# B&R Automation Studio project NAEUL004C00R13L518F00 (part 19)

#### Act_OptP0931MagConv2FB.st
```iecst
ACTION Act_OptP0931MagConv2FB:

	//Magazine Conveyor
	IF tyP0931MagConv2.tyFB.tyBtnStop.bRtCompl = TRUE THEN
		eMagConv2Clp2Act	:= MagConv2ClpActStop;

		IF p_eMagConv2Clp2Stat = MagConv2ClpActStop AND p_eMagConv2Clp2Status = Done THEN
			eMagConv2Clp2Act	:= MagConv2ClpActIdle;

			tyP0931MagConv2.tyFB.tyBtnEnt.bRtCompl	:= FALSE;
			tyP0931MagConv2.tyFB.tyBtnEnt.bValue	:= FALSE;
			tyP0931MagConv2.tyFB.tyBtnEnt.bRtLk		:= FALSE;

			tyP0931MagConv2.tyFB.tyBtnExit.bRtCompl	:= FALSE;
			tyP0931MagConv2.tyFB.tyBtnExit.bValue	:= FALSE;
			tyP0931MagConv2.tyFB.tyBtnExit.bRtLk	:= FALSE;

			tyP0931MagConv2.tyFB.tyBtnStop.bRtCompl	:= FALSE;
			tyP0931MagConv2.tyFB.tyBtnStop.bValue	:= TRUE;
			tyP0931MagConv2.tyFB.tyBtnStop.bRtLk	:= TRUE;
		END_IF

	ELSIF tyP0931MagConv2.tyFB.tyBtnEnt.bRtCompl = TRUE THEN
		tyP0931MagConv2.tyFB.tyBtnEnt.bValue	:= TRUE;
		tyP0931MagConv2.tyFB.tyBtnEnt.bRtLk		:= TRUE;

		tyP0931MagConv2.tyFB.tyBtnStop.bValue	:= FALSE;
		tyP0931MagConv2.tyFB.tyBtnStop.bRtLk	:= FALSE;

		eMagConv2Clp2Act	:= MagConv2ClpActEnt;

		IF p_eMagConv2Clp2Stat = MagConv2ClpActEnt AND p_eMagConv2Clp2Status = Done THEN
			eMagConv2Clp2Act	:= MagConv2ClpActIdle;

			tyP0931MagConv2.tyFB.tyBtnEnt.bRtCompl	:= FALSE;

			tyP0931MagConv2.tyFB.tyBtnEnt.bValue	:= FALSE;
			tyP0931MagConv2.tyFB.tyBtnEnt.bRtLk		:= FALSE;

			tyP0931MagConv2.tyFB.tyBtnStop.bValue	:= TRUE;
			tyP0931MagConv2.tyFB.tyBtnStop.bRtLk	:= TRUE;
		END_IF

	ELSIF (p_eMagConv2Clp2Stat = MagConv2ClpActPreExit AND p_eMagConv2Clp2Status = Done) THEN
		eMagConv2Clp2Act	:= MagConv2ClpActIdle;

		tyP0931MagConv2.tyFB.tyBtnExit.bRtCompl	:= FALSE;

		tyP0931MagConv2.tyFB.tyBtnExit.bValue	:= FALSE;
		tyP0931MagConv2.tyFB.tyBtnExit.bRtLk	:= FALSE;

		tyP0931MagConv2.tyFB.tyBtnStop.bValue	:= TRUE;
		tyP0931MagConv2.tyFB.tyBtnStop.bRtLk	:= TRUE;

	ELSIF (p_eMagConv2Clp2Stat = MagConv2ClpActExit AND p_eMagConv2Clp2Status = Done) THEN
		eMagConv2Clp2Act	:= MagConv2ClpActIdle;

		tyP0931MagConv2.tyFB.tyBtnExit.bRtCompl	:= FALSE;

		tyP0931MagConv2.tyFB.tyBtnExit.bValue	:= FALSE;
		tyP0931MagConv2.tyFB.tyBtnExit.bRtLk	:= FALSE;

		tyP0931MagConv2.tyFB.tyBtnStop.bValue	:= TRUE;
		tyP0931MagConv2.tyFB.tyBtnStop.bRtLk	:= TRUE;

	ELSIF tyP0931MagConv2.tyFB.tyBtnExit.bRtCompl = TRUE THEN
		tyP0931MagConv2.tyFB.tyBtnExit.bRtCompl	:= FALSE;
		tyP0931MagConv2.tyFB.tyBtnExit.bValue	:= TRUE;
		tyP0931MagConv2.tyFB.tyBtnExit.bRtLk	:= TRUE;

		tyP0931MagConv2.tyFB.tyBtnStop.bValue	:= FALSE;
		tyP0931MagConv2.tyFB.tyBtnStop.bRtLk	:= FALSE;

		IF p_tyDI.bMagConvEntSen2  THEN
			eMagConv2Clp2Act	:= MagConv2ClpActExit;
		ELSE
			IF p_tyDI.bMagPresentSen2 THEN
				eMagConv2Clp2Act	:= MagConv2ClpActPreExit;
			ELSE
				eMagConv2Clp2Act	:= MagConv2ClpActExit;
			END_IF
		END_IF
	END_IF

	//Magazine Clamper
	IF tyP0931MagConv2.tyCom.tyBtnSwitch.bValue = FALSE THEN

		//Fixed
		IF tyP0931MagConv2.tyFB.tyBtnFixedUnclamp.bRtCompl = TRUE THEN
			tyP0931MagConv2.tyFB.tyBtnFixedUnclamp.bRtCompl	:= FALSE;

			tyP0931MagConv2.tyFB.tyBtnFixedUnclamp.bValue	:= TRUE;
			tyP0931MagConv2.tyFB.tyBtnFixedClamp.bValue		:= FALSE;

		ELSIF tyP0931MagConv2.tyFB.tyBtnFixedClamp.bRtCompl = TRUE THEN
			tyP0931MagConv2.tyFB.tyBtnFixedClamp.bRtCompl	:= FALSE;

			tyP0931MagConv2.tyFB.tyBtnFixedClamp.bValue		:= TRUE;
			tyP0931MagConv2.tyFB.tyBtnFixedUnclamp.bValue	:= FALSE;

		END_IF

		//Remote
		IF tyP0931MagConv2.tyFB.tyBtnRemoteUnclamp.bRtCompl = TRUE THEN
			tyP0931MagConv2.tyFB.tyBtnRemoteUnclamp.bRtCompl	:= FALSE;

			tyP0931MagConv2.tyFB.tyBtnRemoteUnclamp.bValue	:= TRUE;
			tyP0931MagConv2.tyFB.tyBtnRemoteClamp.bValue	:= FALSE;

		ELSIF tyP0931MagConv2.tyFB.tyBtnRemoteClamp.bRtCompl = TRUE THEN
			tyP0931MagConv2.tyFB.tyBtnRemoteClamp.bRtCompl	:= FALSE;

			tyP0931MagConv2.tyFB.tyBtnRemoteClamp.bValue	:= TRUE;
			tyP0931MagConv2.tyFB.tyBtnRemoteUnclamp.bValue	:= FALSE;

		END_IF

		//Selection
		IF tyP0931MagConv2.tyFB.tyBtnSelUnclamp.bRtCompl = TRUE THEN
			tyP0931MagConv2.tyFB.tyBtnSelUnclamp.bRtCompl	:= FALSE;

			tyP0931MagConv2.tyFB.tyBtnSelUnclamp.bValue	:= TRUE;
			tyP0931MagConv2.tyFB.tyBtnSelClamp.bValue	:= FALSE;

		ELSIF tyP0931MagConv2.tyFB.tyBtnSelClamp.bRtCompl = TRUE THEN
			tyP0931MagConv2.tyFB.tyBtnSelClamp.bRtCompl	:= FALSE;

			tyP0931MagConv2.tyFB.tyBtnSelClamp.bValue	:= TRUE;
			tyP0931MagConv2.tyFB.tyBtnSelUnclamp.bValue	:= FALSE;

		END_IF

		// Fixed Clamper
		IF tyP0931MagConv2.tyFB.tyBtnFixedUnclamp.bValue = TRUE THEN

			eMagConv2Clp2Act	:= MagConv2ClpActFixClprUnclamp;

			IF p_eMagConv2Clp2Stat = MagConv2ClpActFixClprUnclamp AND p_eMagConv2Clp2Status = Done THEN

				eMagConv2Clp2Act	:= MagConv2ClpActIdle;

				tyP0931MagConv2.tyFB.tyBtnFixedUnclamp.bValue	:= FALSE;

			ELSIF p_eMagConv2Clp2Status = Error THEN

				tyP0931MagConv2.tyFB.tyBtnFixedUnclamp.bValue	:= FALSE;

			END_IF

		ELSIF tyP0931MagConv2.tyFB.tyBtnFixedClamp.bValue = TRUE THEN
			eMagConv2Clp2Act	:= MagConv2ClpActFixClprClamp;

			IF p_eMagConv2Clp2Stat = MagConv2ClpActFixClprClamp AND p_eMagConv2Clp2Status = Done THEN

				eMagConv2Clp2Act	:= MagConv2ClpActIdle;

				tyP0931MagConv2.tyFB.tyBtnFixedClamp.bValue := FALSE;

			ELSIF p_eMagConv2Clp2Status = Error THEN
				tyP0931MagConv2.tyFB.tyBtnFixedClamp.bValue := FALSE;

			END_IF

		END_IF

		//Remote Clamper
		IF tyP0931MagConv2.tyFB.tyBtnRemoteUnclamp.bValue = TRUE THEN

			eMagConv2Clp2Act	:= MagConv2ClpActRmtClprUnclamp;

			IF p_eMagConv2Clp2Stat = MagConv2ClpActRmtClprUnclamp AND p_eMagConv2Clp2Status = Done THEN

				eMagConv2Clp2Act	:= MagConv2ClpActIdle;

				tyP0931MagConv2.tyFB.tyBtnRemoteUnclamp.bValue	:= FALSE;

			ELSIF p_eMagConv2Clp2Status = Error THEN

				tyP0931MagConv2.tyFB.tyBtnRemoteUnclamp.bValue	:= FALSE;

			END_IF

		ELSIF tyP0931MagConv2.tyFB.tyBtnRemoteClamp.bValue = TRUE THEN
			eMagConv2Clp2Act	:= MagConv2ClpActRmtClprClamp;

			IF p_eMagConv2Clp2Stat = MagConv2ClpActRmtClprClamp AND p_eMagConv2Clp2Status = Done THEN

				eMagConv2Clp2Act	:= MagConv2ClpActIdle;

				tyP0931MagConv2.tyFB.tyBtnRemoteClamp.bValue := FALSE;

			ELSIF p_eMagConv2Clp2Status = Error THEN
				tyP0931MagConv2.tyFB.tyBtnRemoteClamp.bValue := FALSE;

			END_IF

		END_IF

		//Selection Clamper
		IF tyP0931MagConv2.tyFB.tyBtnSelUnclamp.bValue = TRUE THEN

			eMagConvSelClp2Act	:= PneuActExt;

			IF p_eSelClamp2Stat = PneuActExt AND p_eSelClamp2Status = Done THEN

				eMagConvSelClp2Act	:= PneuActIdle;

				tyP0931MagConv2.tyFB.tyBtnSelUnclamp.bValue	:= FALSE;

			ELSIF p_eSelClamp2Status = Error THEN

				tyP0931MagConv2.tyFB.tyBtnSelUnclamp.bValue	:= FALSE;

			END_IF

		ELSIF tyP0931MagConv2.tyFB.tyBtnSelClamp.bValue = TRUE THEN
			eMagConvSelClp2Act	:= PneuActRet;

			IF p_eSelClamp2Stat = PneuActRet AND p_eSelClamp2Status = Done THEN

				eMagConvSelClp2Act	:= PneuActIdle;

				tyP0931MagConv2.tyFB.tyBtnSelClamp.bValue	:= FALSE;

			ELSIF p_eSelClamp2Status = Error THEN
				tyP0931MagConv2.tyFB.tyBtnSelClamp.bValue	:= FALSE;

			END_IF

		END_IF

		//Update Status
		tyP0931MagConv2.tyDC.tyBtnFixedUnclamp.bValue	:= NOT p_bMagConv2Clp2ClprFixClampCtrl;
		tyP0931MagConv2.tyDC.tyBtnFixedClamp.bValue		:= p_bMagConv2Clp2ClprFixClampCtrl;
		tyP0931MagConv2.tyDC.tyBtnRemoteUnclamp.bValue	:= NOT p_bMagConv2Clp2ClprRmtClampCtrl;
		tyP0931MagConv2.tyDC.tyBtnRemoteClamp.bValue	:= p_bMagConv2Clp2ClprRmtClampCtrl;

		tyP0931MagConv2.tyDC.tyBtnSelUnclamp.bRtCompl	:= FALSE;
		tyP0931MagConv2.tyDC.tyBtnSelClamp.bRtCompl		:= FALSE;
		tyP0931MagConv2.tyDC.tyBtnSelUnclamp.bValue	:= p_bSelClamp2RetCtrl;
		tyP0931MagConv2.tyDC.tyBtnSelClamp.bValue	:= p_bSelClamp2ExtCtrl;
	END_IF

	//Mask
	IF p_tyUsrMgmtCurrAccessRgt.bManualFBOnly THEN

		fUIInRtStatOff(ADR(tyP0931MagConv2.tyCom.tyBtnSwitch.uiMaskRtStat));

	ELSE

	IF p_eMagConv2Clp2Status = Error THEN

		fUIInRtStatOff(ADR(tyP0931MagConv2.tyFB.tyBtnEnt.uiMaskRtStat));
		fUIInRtStatOff(ADR(tyP0931MagConv2.tyFB.tyBtnExit.uiMaskRtStat));
		fUIInRtStatOff(ADR(tyP0931MagConv2.tyFB.tyBtnFixedClamp.uiMaskRtStat));
		fUIInRtStatOff(ADR(tyP0931MagConv2.tyFB.tyBtnFixedUnclamp.uiMaskRtStat));
		fUIInRtStatOff(ADR(tyP0931MagConv2.tyFB.tyBtnRemoteClamp.uiMaskRtStat));
		fUIInRtStatOff(ADR(tyP0931MagConv2.tyFB.tyBtnRemoteUnclamp.uiMaskRtStat));
			fUIInRtStatOff(ADR(tyP0931MagConv2.tyFB.tyBtnSelClamp.uiMaskRtStat));
			fUIInRtStatOff(ADR(tyP0931MagConv2.tyFB.tyBtnSelUnclamp.uiMaskRtStat));
		fUIInRtStatHide(ADR(tyP0931MagConv2.tyCom.tyBtnSwitch.uiMaskRtStat));

	ELSIF tyP0931MagConv2.tyFB.tyBtnEnt.bRtCompl = TRUE THEN

		fUIInRtStatHide(ADR(tyP0931MagConv2.tyFB.tyBtnEnt.uiMaskRtStat));
		fUIInRtStatOff(ADR(tyP0931MagConv2.tyFB.tyBtnExit.uiMaskRtStat));
		fUIInRtStatOff(ADR(tyP0931MagConv2.tyFB.tyBtnFixedClamp.uiMaskRtStat));
		fUIInRtStatOff(ADR(tyP0931MagConv2.tyFB.tyBtnFixedUnclamp.uiMaskRtStat));
		fUIInRtStatOff(ADR(tyP0931MagConv2.tyFB.tyBtnRemoteClamp.uiMaskRtStat));
		fUIInRtStatOff(ADR(tyP0931MagConv2.tyFB.tyBtnRemoteUnclamp.uiMaskRtStat));
			fUIInRtStatOff(ADR(tyP0931MagConv2.tyFB.tyBtnSelClamp.uiMaskRtStat));
			fUIInRtStatOff(ADR(tyP0931MagConv2.tyFB.tyBtnSelUnclamp.uiMaskRtStat));
		fUIInRtStatOff(ADR(tyP0931MagConv2.tyCom.tyBtnSwitch.uiMaskRtStat));

	ELSIF tyP0931MagConv2.tyFB.tyBtnExit.bRtCompl = TRUE THEN

		fUIInRtStatOff(ADR(tyP0931MagConv2.tyFB.tyBtnEnt.uiMaskRtStat));
		fUIInRtStatHide(ADR(tyP0931MagConv2.tyFB.tyBtnExit.uiMaskRtStat));
		fUIInRtStatOff(ADR(tyP0931MagConv2.tyFB.tyBtnFixedClamp.uiMaskRtStat));
		fUIInRtStatOff(ADR(tyP0931MagConv2.tyFB.tyBtnFixedUnclamp.uiMaskRtStat));
		fUIInRtStatOff(ADR(tyP0931MagConv2.tyFB.tyBtnRemoteClamp.uiMaskRtStat));
		fUIInRtStatOff(ADR(tyP0931MagConv2.tyFB.tyBtnRemoteUnclamp.uiMaskRtStat));
		fUIInRtStatOff(ADR(tyP0931MagConv2.tyFB.tyBtnSelClamp.uiMaskRtStat));
		fUIInRtStatOff(ADR(tyP0931MagConv2.tyFB.tyBtnSelUnclamp.uiMaskRtStat));
		fUIInRtStatOff(ADR(tyP0931MagConv2.tyCom.tyBtnSwitch.uiMaskRtStat));

	ELSIF tyP0931MagConv2.tyFB.tyBtnFixedClamp.bValue = TRUE OR tyP0931MagConv2.tyFB.tyBtnRemoteClamp.bValue = TRUE
			OR tyP0931MagConv2.tyFB.tyBtnFixedUnclamp.bValue = TRUE OR tyP0931MagConv2.tyFB.tyBtnRemoteUnclamp.bValue = TRUE
			OR tyP0931MagConv2.tyFB.tyBtnSelClamp.bValue = TRUE OR tyP0931MagConv2.tyFB.tyBtnSelUnclamp.bValue = TRUE
			THEN

		fUIInRtStatOff(ADR(tyP0931MagConv2.tyFB.tyBtnEnt.uiMaskRtStat));
		fUIInRtStatOff(ADR(tyP0931MagConv2.tyFB.tyBtnExit.uiMaskRtStat));
		fUIInRtStatHide(ADR(tyP0931MagConv2.tyFB.tyBtnFixedClamp.uiMaskRtStat));
		fUIInRtStatHide(ADR(tyP0931MagConv2.tyFB.tyBtnFixedUnclamp.uiMaskRtStat));
		fUIInRtStatHide(ADR(tyP0931MagConv2.tyFB.tyBtnRemoteClamp.uiMaskRtStat));
		fUIInRtStatHide(ADR(tyP0931MagConv2.tyFB.tyBtnRemoteUnclamp.uiMaskRtStat));
		fUIInRtStatHide(ADR(tyP0931MagConv2.tyFB.tyBtnSelClamp.uiMaskRtStat));
		fUIInRtStatHide(ADR(tyP0931MagConv2.tyFB.tyBtnSelUnclamp.uiMaskRtStat));
		fUIInRtStatOff(ADR(tyP0931MagConv2.tyCom.tyBtnSwitch.uiMaskRtStat));

	ELSE

		fUIInRtStatHide(ADR(tyP0931MagConv2.tyFB.tyBtnEnt.uiMaskRtStat));
		fUIInRtStatHide(ADR(tyP0931MagConv2.tyFB.tyBtnExit.uiMaskRtStat));
		fUIInRtStatHide(ADR(tyP0931MagConv2.tyFB.tyBtnFixedClamp.uiMaskRtStat));
		fUIInRtStatHide(ADR(tyP0931MagConv2.tyFB.tyBtnFixedUnclamp.uiMaskRtStat));
		fUIInRtStatHide(ADR(tyP0931MagConv2.tyFB.tyBtnRemoteClamp.uiMaskRtStat));
		fUIInRtStatHide(ADR(tyP0931MagConv2.tyFB.tyBtnRemoteUnclamp.uiMaskRtStat));
		fUIInRtStatHide(ADR(tyP0931MagConv2.tyFB.tyBtnSelClamp.uiMaskRtStat));
		fUIInRtStatHide(ADR(tyP0931MagConv2.tyFB.tyBtnSelUnclamp.uiMaskRtStat));
		fUIInRtStatHide(ADR(tyP0931MagConv2.tyCom.tyBtnSwitch.uiMaskRtStat));

	END_IF
END_IF

	IF p_tyDI.bMagConvCAB717MagSen2 THEN
		fUIInRtStatOff(ADR(tyP0931MagConv2.tyFB.tyBtnSelClamp.uiMaskRtStat));
	END_IF

	IF p_bMagConv2Clp2ClprFixClampCtrl OR p_bMagConv2Clp2ClprRmtClampCtrl THEN
		fUIInRtStatOff(ADR(tyP0931MagConv2.tyFB.tyBtnEnt.uiMaskRtStat));
		fUIInRtStatOff(ADR(tyP0931MagConv2.tyFB.tyBtnExit.uiMaskRtStat));
	END_IF

END_ACTION
```

#### Act_OptP0931MagConv2FBStat.st
```iecst
ACTION Act_OptP0931MagConv2FBStat:

	IF tyP0931MagConv2.tyFB.tyBtnFixedClamp.bValue = TRUE OR tyP0931MagConv2.tyFB.tyBtnRemoteClamp.bValue = TRUE
		OR tyP0931MagConv2.tyFB.tyBtnFixedUnclamp.bValue = TRUE OR tyP0931MagConv2.tyFB.tyBtnRemoteUnclamp.bValue = TRUE
		THEN
		tyP0931MagConv2.tyFB.tyStringStat.sValue	:= p_sMagConv2Clp2StatTxt;

	ELSIF (tyP0931MagConv2.tyFB.tyBtnFixedClamp.bValue = FALSE AND  tyP0931MagConv2.tyFB.tyBtnRemoteClamp.bValue = FALSE
		AND tyP0931MagConv2.tyFB.tyBtnFixedUnclamp.bValue = FALSE AND  tyP0931MagConv2.tyFB.tyBtnRemoteUnclamp.bValue = FALSE
		AND p_eMagConv2Clp2Status <> Busy )
		THEN
		tyP0931MagConv2.tyFB.tyStringStat.sValue	:= p_sMagConv2Clp2StatTxt;

	ELSIF tyP0931MagConv2.tyFB.tyBtnSelUnclamp.bValue = TRUE OR tyP0931MagConv2.tyFB.tyBtnSelClamp.bValue = TRUE
		THEN
		tyP0931MagConv2.tyFB.tyStringStat.sValue	:= p_sSelClamp2StatTxt;
	END_IF
END_ACTION
```

#### Act_OptP0931MagConv2DC.st
```iecst
ACTION Act_OptP0931MagConv2DC:

	//Magazine Conveyor
	IF tyP0931MagConv2.tyDC.tyBtnStop.bRtCompl = TRUE THEN
		eMagConv2Clp2Act	:= MagConv2ClpActStop;

		IF p_eMagConv2Clp2Stat = MagConv2ClpActStop AND p_eMagConv2Clp2Status = Done THEN
			eMagConv2Clp2Act	:= MagConv2ClpActIdle;

			tyP0931MagConv2.tyDC.tyBtnStop.bRtCompl		:= FALSE;
			tyP0931MagConv2.tyDC.tyBtnStop.bValue		:= TRUE;
			tyP0931MagConv2.tyDC.tyBtnStop.bRtLk		:= TRUE;

			tyP0931MagConv2.tyDC.tyBtnMagIn.bRtCompl	:= FALSE;
			tyP0931MagConv2.tyDC.tyBtnMagIn.bValue		:= FALSE;
			tyP0931MagConv2.tyDC.tyBtnMagIn.bRtLk		:= FALSE;

			tyP0931MagConv2.tyDC.tyBtnMagOut.bRtCompl	:= FALSE;
			tyP0931MagConv2.tyDC.tyBtnMagOut.bValue		:= FALSE;
			tyP0931MagConv2.tyDC.tyBtnMagOut.bRtLk		:= FALSE;
		END_IF

	ELSIF tyP0931MagConv2.tyDC.tyBtnMagIn.bRtCompl = TRUE THEN
		tyP0931MagConv2.tyDC.tyBtnMagIn.bValue	:= TRUE;
		tyP0931MagConv2.tyDC.tyBtnMagIn.bRtLk	:= TRUE;

		tyP0931MagConv2.tyDC.tyBtnStop.bValue	:= FALSE;
		tyP0931MagConv2.tyDC.tyBtnStop.bRtLk	:= FALSE;

		IF p_tyNtParamCurr.eProjMagConvDir = ConvDirLToR OR p_tyNtParamCurr.eProjMagConvDir = ConvDirLToL THEN

			eMagConv2Clp2Act	:= MagConv2ClpActSetMtrSigOnOrLToR;

			IF p_eMagConv2Clp2Stat = MagConv2ClpActSetMtrSigOnOrLToR AND p_eMagConv2Clp2Status = Done THEN
				eMagConv2Clp2Act	:= MagConv2ClpActIdle;

				tyP0931MagConv2.tyDC.tyBtnMagIn.bRtCompl	:= FALSE;
			END_IF

		ELSE

			eMagConv2Clp2Act	:= MagConv2ClpActSetMtrDirOrRToL;

			IF p_eMagConv2Clp2Stat = MagConv2ClpActSetMtrDirOrRToL AND p_eMagConv2Clp2Status = Done THEN
				eMagConv2Clp2Act	:= MagConv2ClpActIdle;

				tyP0931MagConv2.tyDC.tyBtnMagIn.bRtCompl	:= FALSE;
			END_IF

		END_IF

	ELSIF tyP0931MagConv2.tyDC.tyBtnMagOut.bRtCompl = TRUE THEN
		tyP0931MagConv2.tyDC.tyBtnMagOut.bValue	:= TRUE;
		tyP0931MagConv2.tyDC.tyBtnMagOut.bRtLk	:= TRUE;

		tyP0931MagConv2.tyDC.tyBtnStop.bValue	:= FALSE;
		tyP0931MagConv2.tyDC.tyBtnStop.bRtLk	:= FALSE;

		IF p_tyNtParamCurr.eProjMagConvDir = ConvDirLToR OR p_tyNtParamCurr.eProjMagConvDir = ConvDirRToR THEN

			eMagConv2Clp2Act	:= MagConv2ClpActSetMtrSigOnOrLToR;

			IF p_eMagConv2Clp2Stat = MagConv2ClpActSetMtrSigOnOrLToR AND p_eMagConv2Clp2Status = Done THEN
				eMagConv2Clp2Act	:= MagConv2ClpActIdle;

				tyP0931MagConv2.tyDC.tyBtnMagOut.bRtCompl	:= FALSE;
			END_IF

		ELSE

			eMagConv2Clp2Act	:= MagConv2ClpActSetMtrDirOrRToL;

			IF p_eMagConv2Clp2Stat = MagConv2ClpActSetMtrDirOrRToL AND p_eMagConv2Clp2Status = Done THEN
				eMagConv2Clp2Act	:= MagConv2ClpActIdle;

				tyP0931MagConv2.tyDC.tyBtnMagOut.bRtCompl	:= FALSE;
			END_IF

		END_IF

	END_IF

	//Magazine Clamper
	IF tyP0931MagConv2.tyCom.tyBtnSwitch.bValue = TRUE THEN
		IF p_bSelClamp2TwoCtrlOut = FALSE THEN
			IF tyP0931MagConv2.tyDC.tyBtnSelUnclamp.bRtCompl = TRUE THEN
				tyP0931MagConv2.tyDC.tyBtnSelUnclamp.bValue := TRUE;
				tyP0931MagConv2.tyDC.tyBtnSelClamp.bValue := FALSE;

				eMagConvSelClp2Act	:= PneuActSetExt;

				IF p_eSelClamp2Stat = PneuActSetExt AND p_eSelClamp2Status = Done THEN
					eMagConvSelClp2Act	:= PneuActIdle;

					tyP0931MagConv2.tyDC.tyBtnSelUnclamp.bRtCompl	:= FALSE;
				END_IF

			ELSIF tyP0931MagConv2.tyDC.tyBtnSelClamp.bRtCompl = TRUE THEN
				tyP0931MagConv2.tyDC.tyBtnSelClamp.bValue := TRUE;
				tyP0931MagConv2.tyDC.tyBtnSelUnclamp.bValue := FALSE;

				eMagConvSelClp2Act	:= PneuActSetRet;

				IF p_eSelClamp2Stat = PneuActSetRet AND p_eSelClamp2Status = Done THEN
					eMagConvSelClp2Act	:= PneuActIdle;

					tyP0931MagConv2.tyDC.tyBtnSelClamp.bRtCompl	:= FALSE;
				END_IF
			END_IF

		ELSE
			IF (tyP0931MagConv2.tyDC.tyBtnSelUnclamp.bRtCompl = TRUE) OR (tyP0931MagConv2.tyDC.tyBtnSelClamp.bRtCompl = TRUE) THEN
				IF (tyP0931MagConv2.tyDC.tyBtnSelUnclamp.bValue = TRUE) AND (tyP0931MagConv2.tyDC.tyBtnSelClamp.bValue = TRUE) THEN
					eMagConvSelClp2Act	:= PneuActSetAll;

					IF p_eSelClamp2Stat = PneuActSetAll AND p_eSelClamp2Status = Done THEN
						eMagConvSelClp2Act	:= PneuActIdle;

						tyP0931MagConv2.tyDC.tyBtnSelUnclamp.bRtCompl		:= FALSE;
						tyP0931MagConv2.tyDC.tyBtnSelClamp.bRtCompl			:= FALSE;
					END_IF

				ELSIF (tyP0931MagConv2.tyDC.tyBtnSelUnclamp.bValue = TRUE) AND (tyP0931MagConv2.tyDC.tyBtnSelClamp.bValue = FALSE) THEN
					eMagConvSelClp2Act	:= PneuActSetExt;

					IF p_eSelClamp2Stat = PneuActSetExt AND p_eSelClamp2Status = Done THEN
						eMagConvSelClp2Act	:= PneuActIdle;

						tyP0931MagConv2.tyDC.tyBtnSelUnclamp.bRtCompl		:= FALSE;
						tyP0931MagConv2.tyDC.tyBtnSelClamp.bRtCompl			:= FALSE;
					END_IF

				ELSIF (tyP0931MagConv2.tyDC.tyBtnSelUnclamp.bValue = FALSE) AND (tyP0931MagConv2.tyDC.tyBtnSelClamp.bValue = TRUE) THEN
					eMagConvSelClp2Act	:= PneuActSetRet;

					IF p_eSelClamp2Stat = PneuActSetRet AND p_eSelClamp2Status = Done THEN
						eMagConvSelClp2Act	:= PneuActIdle;

						tyP0931MagConv2.tyDC.tyBtnSelUnclamp.bRtCompl		:= FALSE;
						tyP0931MagConv2.tyDC.tyBtnSelClamp.bRtCompl			:= FALSE;
					END_IF

				ELSE
					eMagConvSelClp2Act	:= PneuActRstAll;

					IF p_eSelClamp2Stat = PneuActRstAll AND p_eSelClamp2Status = Done THEN
						eMagConvSelClp2Act	:= PneuActIdle;

						tyP0931MagConv2.tyDC.tyBtnSelUnclamp.bRtCompl		:= FALSE;
						tyP0931MagConv2.tyDC.tyBtnSelClamp.bRtCompl			:= FALSE;
					END_IF

				END_IF
			END_IF
		END_IF

			IF p_bMagConv2Clp1ClprTwoOutputCtrl = FALSE THEN

				IF tyP0931MagConv2.tyDC.tyBtnFixedClamp.bRtCompl = TRUE THEN
					tyP0931MagConv2.tyDC.tyBtnFixedClamp.bValue		:= TRUE;
					tyP0931MagConv2.tyDC.tyBtnFixedUnclamp.bValue	:= FALSE;

					eMagConv2Clp2Act	:= MagConv2ClpActFixClprSetClamp;

					IF p_eMagConv2Clp2Stat = MagConv2ClpActFixClprSetClamp AND p_eMagConv2Clp2Status = Done THEN
						eMagConv2Clp2Act	:= MagConv2ClpActIdle;

						tyP0931MagConv2.tyDC.tyBtnFixedClamp.bRtCompl	:= FALSE;
					END_IF

				ELSIF tyP0931MagConv2.tyDC.tyBtnFixedUnclamp.bRtCompl = TRUE THEN
					tyP0931MagConv2.tyDC.tyBtnFixedUnclamp.bValue	:= TRUE;
					tyP0931MagConv2.tyDC.tyBtnFixedClamp.bValue		:= FALSE;

					eMagConv2Clp2Act	:= MagConv2ClpActFixClprSetUnclamp;

					IF p_eMagConv2Clp2Stat = MagConv2ClpActFixClprSetUnclamp AND p_eMagConv2Clp2Status = Done THEN
						eMagConv2Clp2Act	:= MagConv2ClpActIdle;

						tyP0931MagConv2.tyDC.tyBtnFixedUnclamp.bRtCompl	:= FALSE;
					END_IF

				END_IF

				//Remote
				IF tyP0931MagConv2.tyDC.tyBtnRemoteClamp.bRtCompl = TRUE THEN
					tyP0931MagConv2.tyDC.tyBtnRemoteClamp.bValue		:= TRUE;
					tyP0931MagConv2.tyDC.tyBtnRemoteUnclamp.bValue		:= FALSE;

					eMagConv2Clp2Act	:= MagConv2ClpActRmtClprSetClamp;

					IF p_eMagConv2Clp2Stat = MagConv2ClpActRmtClprSetClamp AND p_eMagConv2Clp2Status = Done THEN
						eMagConv2Clp2Act	:= MagConv2ClpActIdle;

						tyP0931MagConv2.tyDC.tyBtnRemoteClamp.bRtCompl	:= FALSE;
					END_IF

				ELSIF tyP0931MagConv2.tyDC.tyBtnRemoteUnclamp.bRtCompl = TRUE THEN
					tyP0931MagConv2.tyDC.tyBtnRemoteUnclamp.bValue	:= TRUE;
					tyP0931MagConv2.tyDC.tyBtnRemoteClamp.bValue	:= FALSE;

					eMagConv2Clp2Act	:= MagConv2ClpActRmtClprSetUnclamp;

					IF p_eMagConv2Clp2Stat = MagConv2ClpActRmtClprSetUnclamp AND p_eMagConv2Clp2Status = Done THEN
						eMagConv2Clp2Act	:= MagConv2ClpActIdle;

						tyP0931MagConv2.tyDC.tyBtnRemoteUnclamp.bRtCompl	:= FALSE;
					END_IF

				END_IF

			ELSE

				//Fixed
				IF (tyP0931MagConv2.tyDC.tyBtnFixedClamp.bRtCompl = TRUE) OR (tyP0931MagConv2.tyDC.tyBtnFixedUnclamp.bRtCompl = TRUE) THEN

					IF (tyP0931MagConv2.tyDC.tyBtnFixedClamp.bValue = TRUE) AND (tyP0931MagConv2.tyDC.tyBtnFixedUnclamp.bValue = TRUE) THEN

						eMagConv2Clp2Act	:= MagConv2ClpActFixClprSetAll;

						IF p_eMagConv2Clp2Stat = MagConv2ClpActFixClprSetAll AND p_eMagConv2Clp2Status = Done THEN

							eMagConv2Clp2Act	:= MagConv2ClpActIdle;

							tyP0931MagConv2.tyDC.tyBtnFixedClamp.bRtCompl	:= FALSE;
						tyP0931MagConv2.tyDC.tyBtnFixedUnclamp.bRtCompl	:= FALSE;
					END_IF

				ELSIF (tyP0931MagConv2.tyDC.tyBtnFixedClamp.bValue = TRUE) AND (tyP0931MagConv2.tyDC.tyBtnFixedUnclamp.bValue = FALSE) THEN
					eMagConv2Clp2Act	:= MagConv2ClpActFixClprSetClamp;

					IF p_eMagConv2Clp2Stat = MagConv2ClpActFixClprSetClamp AND p_eMagConv2Clp2Status = Done THEN

						eMagConv2Clp2Act	:= MagConv2ClpActIdle;

						tyP0931MagConv2.tyDC.tyBtnFixedClamp.bRtCompl	:= FALSE;
						tyP0931MagConv2.tyDC.tyBtnFixedUnclamp.bRtCompl	:= FALSE;
					END_IF

				ELSIF (tyP0931MagConv2.tyDC.tyBtnFixedClamp.bValue = FALSE) AND (tyP0931MagConv2.tyDC.tyBtnFixedUnclamp.bValue = TRUE) THEN
					eMagConv2Clp2Act	:= MagConv2ClpActFixClprSetUnclamp;

					IF p_eMagConv2Clp2Stat = MagConv2ClpActFixClprSetUnclamp AND p_eMagConv2Clp2Status = Done THEN

						eMagConv2Clp2Act	:= MagConv2ClpActIdle;

						tyP0931MagConv2.tyDC.tyBtnFixedClamp.bRtCompl	:= FALSE;
						tyP0931MagConv2.tyDC.tyBtnFixedUnclamp.bRtCompl	:= FALSE;
					END_IF

				ELSE
					eMagConv2Clp2Act	:= MagConv2ClpActFixClprRstAll;

					IF p_eMagConv2Clp2Stat = MagConv2ClpActFixClprRstAll AND p_eMagConv2Clp2Status = Done THEN

						eMagConv2Clp2Act	:= MagConv2ClpActIdle;

						tyP0931MagConv2.tyDC.tyBtnFixedClamp.bRtCompl	:= FALSE;
						tyP0931MagConv2.tyDC.tyBtnFixedUnclamp.bRtCompl	:= FALSE;
					END_IF

				END_IF

				//Remote
				IF (tyP0931MagConv2.tyDC.tyBtnRemoteClamp.bRtCompl = TRUE) OR (tyP0931MagConv2.tyDC.tyBtnRemoteUnclamp.bRtCompl = TRUE) THEN

					IF (tyP0931MagConv2.tyDC.tyBtnRemoteClamp.bValue = TRUE) AND (tyP0931MagConv2.tyDC.tyBtnRemoteUnclamp.bValue = TRUE) THEN

						eMagConv2Clp2Act	:= MagConv2ClpActRmtClprSetAll;

						IF p_eMagConv2Clp2Stat = MagConv2ClpActRmtClprSetAll AND p_eMagConv2Clp2Status = Done THEN

							eMagConv2Clp2Act	:= MagConv2ClpActIdle;

							tyP0931MagConv2.tyDC.tyBtnRemoteClamp.bRtCompl		:= FALSE;
							tyP0931MagConv2.tyDC.tyBtnRemoteUnclamp.bRtCompl	:= FALSE;
						END_IF

					ELSIF (tyP0931MagConv2.tyDC.tyBtnRemoteClamp.bValue = TRUE) AND (tyP0931MagConv2.tyDC.tyBtnRemoteUnclamp.bValue = FALSE) THEN
						eMagConv2Clp2Act	:= MagConv2ClpActRmtClprSetClamp;

						IF p_eMagConv2Clp2Stat = MagConv2ClpActRmtClprSetClamp AND p_eMagConv2Clp2Status = Done THEN

							eMagConv2Clp2Act	:= MagConv2ClpActIdle;

							tyP0931MagConv2.tyDC.tyBtnRemoteClamp.bRtCompl	:= FALSE;
							tyP0931MagConv2.tyDC.tyBtnRemoteUnclamp.bRtCompl	:= FALSE;
						END_IF

					ELSIF (tyP0931MagConv2.tyDC.tyBtnRemoteClamp.bValue = FALSE) AND (tyP0931MagConv2.tyDC.tyBtnRemoteUnclamp.bValue = TRUE) THEN
						eMagConv2Clp2Act	:= MagConv2ClpActRmtClprSetUnclamp;

						IF p_eMagConv2Clp2Stat = MagConv2ClpActRmtClprSetUnclamp AND p_eMagConv2Clp2Status = Done THEN

							eMagConv2Clp2Act	:= MagConv2ClpActIdle;

							tyP0931MagConv2.tyDC.tyBtnRemoteClamp.bRtCompl	:= FALSE;
							tyP0931MagConv2.tyDC.tyBtnRemoteUnclamp.bRtCompl	:= FALSE;
						END_IF

					ELSE
						eMagConv2Clp2Act	:= MagConv2ClpActRmtClprRstAll;

						IF p_eMagConv2Clp2Stat = MagConv2ClpActRmtClprRstAll AND p_eMagConv2Clp2Status = Done THEN

							eMagConv2Clp2Act	:= MagConv2ClpActIdle;

							tyP0931MagConv2.tyDC.tyBtnRemoteClamp.bRtCompl	:= FALSE;
							tyP0931MagConv2.tyDC.tyBtnRemoteUnclamp.bRtCompl	:= FALSE;
						END_IF

					END_IF
				END_IF

			END_IF

		END_IF

		//Fixed
		tyP0931MagConv2.tyFB.tyBtnFixedClamp.bRtCompl		:= FALSE;
		tyP0931MagConv2.tyFB.tyBtnFixedClamp.bValue			:= FALSE;
		tyP0931MagConv2.tyFB.tyBtnFixedUnclamp.bRtCompl		:= FALSE;
		tyP0931MagConv2.tyFB.tyBtnFixedUnclamp.bValue		:= FALSE;

		//Remote
		tyP0931MagConv2.tyFB.tyBtnRemoteClamp.bRtCompl		:= FALSE;
		tyP0931MagConv2.tyFB.tyBtnRemoteClamp.bValue		:= FALSE;
		tyP0931MagConv2.tyFB.tyBtnRemoteUnclamp.bRtCompl	:= FALSE;
		tyP0931MagConv2.tyFB.tyBtnRemoteUnclamp.bValue		:= FALSE;

	END_IF

	//Mask
	IF p_eMagConv2Clp2Status = Error THEN

		fUIInRtStatOff(ADR(tyP0931MagConv2.tyDC.tyBtnMagIn.uiMaskRtStat));
		fUIInRtStatOff(ADR(tyP0931MagConv2.tyDC.tyBtnMagOut.uiMaskRtStat));
		fUIInRtStatOff(ADR(tyP0931MagConv2.tyDC.tyBtnFixedClamp.uiMaskRtStat));
		fUIInRtStatOff(ADR(tyP0931MagConv2.tyDC.tyBtnFixedUnclamp.uiMaskRtStat));
		fUIInRtStatOff(ADR(tyP0931MagConv2.tyDC.tyBtnRemoteClamp.uiMaskRtStat));
		fUIInRtStatOff(ADR(tyP0931MagConv2.tyDC.tyBtnRemoteUnclamp.uiMaskRtStat));

	ELSIF tyP0931MagConv2.tyDC.tyBtnMagIn.bValue = TRUE THEN

		fUIInRtStatHide(ADR(tyP0931MagConv2.tyDC.tyBtnMagIn.uiMaskRtStat));
		fUIInRtStatOff(ADR(tyP0931MagConv2.tyDC.tyBtnMagOut.uiMaskRtStat));
		fUIInRtStatOff(ADR(tyP0931MagConv2.tyDC.tyBtnFixedClamp.uiMaskRtStat));
		fUIInRtStatOff(ADR(tyP0931MagConv2.tyDC.tyBtnFixedUnclamp.uiMaskRtStat));
		fUIInRtStatOff(ADR(tyP0931MagConv2.tyDC.tyBtnRemoteClamp.uiMaskRtStat));
		fUIInRtStatOff(ADR(tyP0931MagConv2.tyDC.tyBtnRemoteUnclamp.uiMaskRtStat));

	ELSIF tyP0931MagConv2.tyDC.tyBtnMagOut.bValue = TRUE THEN

		fUIInRtStatOff(ADR(tyP0931MagConv2.tyDC.tyBtnMagIn.uiMaskRtStat));
		fUIInRtStatHide(ADR(tyP0931MagConv2.tyDC.tyBtnMagOut.uiMaskRtStat));
		fUIInRtStatOff(ADR(tyP0931MagConv2.tyDC.tyBtnFixedClamp.uiMaskRtStat));
		fUIInRtStatOff(ADR(tyP0931MagConv2.tyDC.tyBtnFixedUnclamp.uiMaskRtStat));
		fUIInRtStatOff(ADR(tyP0931MagConv2.tyDC.tyBtnRemoteClamp.uiMaskRtStat));
		fUIInRtStatOff(ADR(tyP0931MagConv2.tyDC.tyBtnRemoteUnclamp.uiMaskRtStat));

	ELSE

		fUIInRtStatHide(ADR(tyP0931MagConv2.tyDC.tyBtnMagIn.uiMaskRtStat));
		fUIInRtStatHide(ADR(tyP0931MagConv2.tyDC.tyBtnMagOut.uiMaskRtStat));
		fUIInRtStatHide(ADR(tyP0931MagConv2.tyDC.tyBtnFixedClamp.uiMaskRtStat));
		fUIInRtStatHide(ADR(tyP0931MagConv2.tyDC.tyBtnFixedUnclamp.uiMaskRtStat));
		fUIInRtStatHide(ADR(tyP0931MagConv2.tyDC.tyBtnRemoteClamp.uiMaskRtStat));
		fUIInRtStatHide(ADR(tyP0931MagConv2.tyDC.tyBtnRemoteUnclamp.uiMaskRtStat));

	END_IF

END_ACTION
```

#### Act_OptP0931RstMnl.st
```iecst
ACTION Act_OptP0931RstMnl:

	IF EDGEPOS((bManualMod = FALSE) OR (p_eMagConv2Clp2Status = Error)) THEN

		eMagConv2Clp2Act	:= MagConv2ClpActIdle;
		eMagConvSelClp2Act	:= PneuActIdle;
		//Magazine Conveyor
		//FB
		tyP0931MagConv2.tyFB.tyBtnEnt.bRtCompl				:= FALSE;
		tyP0931MagConv2.tyFB.tyBtnExit.bRtCompl				:= FALSE;
		tyP0931MagConv2.tyFB.tyBtnStop.bRtCompl				:= FALSE;

		tyP0931MagConv2.tyFB.tyBtnEnt.bValue				:= FALSE;
		tyP0931MagConv2.tyFB.tyBtnExit.bValue				:= FALSE;
		tyP0931MagConv2.tyFB.tyBtnStop.bValue				:= TRUE;

		tyP0931MagConv2.tyFB.tyBtnEnt.bRtLk					:= FALSE;
		tyP0931MagConv2.tyFB.tyBtnExit.bRtLk				:= FALSE;
		tyP0931MagConv2.tyFB.tyBtnStop.bRtLk				:= TRUE;

		tyP0931MagConv2.tyFB.tyBtnEnt.uiMaskRtStat.0		:= TRUE;
		tyP0931MagConv2.tyFB.tyBtnExit.uiMaskRtStat.0		:= TRUE;
		tyP0931MagConv2.tyCom.tyBtnSwitch.uiMaskRtStat.0	:= TRUE;

		//Direct
		tyP0931MagConv2.tyDC.tyBtnMagIn.bRtCompl			:= FALSE;
		tyP0931MagConv2.tyDC.tyBtnMagOut.bRtCompl			:= FALSE;
		tyP0931MagConv2.tyDC.tyBtnStop.bRtCompl				:= FALSE;

		tyP0931MagConv2.tyDC.tyBtnMagIn.bValue				:= FALSE;
		tyP0931MagConv2.tyDC.tyBtnMagOut.bValue				:= FALSE;
		tyP0931MagConv2.tyDC.tyBtnStop.bValue				:= TRUE;

		tyP0931MagConv2.tyDC.tyBtnMagIn.bRtLk				:= FALSE;
		tyP0931MagConv2.tyDC.tyBtnMagOut.bRtLk				:= FALSE;
		tyP0931MagConv2.tyDC.tyBtnStop.bRtLk				:= TRUE;

		tyP0931MagConv2.tyDC.tyBtnMagIn.uiMaskRtStat.0		:= TRUE;
		tyP0931MagConv2.tyDC.tyBtnMagOut.uiMaskRtStat.0		:= TRUE;
		tyP0931MagConv2.tyCom.tyBtnSwitch.uiMaskRtStat.0	:= TRUE;

		//Magazine Clamper
		//FB
		//Fixed
		tyP0931MagConv2.tyFB.tyBtnFixedClamp.bRtCompl			:= FALSE;
		tyP0931MagConv2.tyFB.tyBtnFixedUnclamp.bRtCompl			:= FALSE;

		tyP0931MagConv2.tyFB.tyBtnFixedClamp.bValue				:= FALSE;
		tyP0931MagConv2.tyFB.tyBtnFixedUnclamp.bValue			:= FALSE;

		//Remote
		tyP0931MagConv2.tyFB.tyBtnRemoteClamp.bRtCompl			:= FALSE;
		tyP0931MagConv2.tyFB.tyBtnRemoteUnclamp.bRtCompl		:= FALSE;

		tyP0931MagConv2.tyFB.tyBtnRemoteClamp.bValue			:= FALSE;
		tyP0931MagConv2.tyFB.tyBtnRemoteUnclamp.bValue			:= FALSE;

		//Selection
		tyP0931MagConv2.tyFB.tyBtnSelClamp.bRtCompl			:= FALSE;
		tyP0931MagConv2.tyFB.tyBtnSelUnclamp.bRtCompl		:= FALSE;

		tyP0931MagConv2.tyFB.tyBtnSelClamp.bValue			:= FALSE;
		tyP0931MagConv2.tyFB.tyBtnSelUnclamp.bValue			:= FALSE;

		tyP0931MagConv2.tyFB.tyBtnFixedClamp.uiMaskRtStat.0		:= TRUE;
		tyP0931MagConv2.tyFB.tyBtnFixedUnclamp.uiMaskRtStat.0	:= TRUE;
		tyP0931MagConv2.tyFB.tyBtnRemoteClamp.uiMaskRtStat.0	:= TRUE;
		tyP0931MagConv2.tyFB.tyBtnRemoteUnclamp.uiMaskRtStat.0	:= TRUE;
		tyP0931MagConv2.tyFB.tyBtnSelClamp.uiMaskRtStat.0		:= TRUE;
		tyP0931MagConv2.tyFB.tyBtnSelUnclamp.uiMaskRtStat.0		:= TRUE;

		tyP0931MagConv2.tyCom.tyBtnSwitch.uiMaskRtStat.0		:= TRUE;

		//Direct
		//Fixed
		tyP0931MagConv2.tyDC.tyBtnFixedClamp.bRtCompl			:= FALSE;
		tyP0931MagConv2.tyDC.tyBtnFixedUnclamp.bRtCompl			:= FALSE;

		tyP0931MagConv2.tyDC.tyBtnFixedClamp.bValue				:= FALSE;
		tyP0931MagConv2.tyDC.tyBtnFixedUnclamp.bValue			:= FALSE;

		//Remote
		tyP0931MagConv2.tyDC.tyBtnRemoteClamp.bRtCompl			:= FALSE;
		tyP0931MagConv2.tyDC.tyBtnRemoteUnclamp.bRtCompl		:= FALSE;

		tyP0931MagConv2.tyDC.tyBtnRemoteClamp.bValue			:= FALSE;
		tyP0931MagConv2.tyDC.tyBtnRemoteUnclamp.bValue			:= FALSE;

		//Selection
		tyP0931MagConv2.tyDC.tyBtnSelClamp.bRtCompl				:= FALSE;
		tyP0931MagConv2.tyDC.tyBtnSelUnclamp.bRtCompl			:= FALSE;

		tyP0931MagConv2.tyDC.tyBtnSelClamp.bValue				:= FALSE;
		tyP0931MagConv2.tyDC.tyBtnSelUnclamp.bValue				:= FALSE;

		tyP0931MagConv2.tyDC.tyBtnFixedClamp.uiMaskRtStat.0		:= TRUE;
		tyP0931MagConv2.tyDC.tyBtnFixedUnclamp.uiMaskRtStat.0	:= TRUE;
		tyP0931MagConv2.tyDC.tyBtnRemoteClamp.uiMaskRtStat.0	:= TRUE;
		tyP0931MagConv2.tyDC.tyBtnRemoteUnclamp.uiMaskRtStat.0	:= TRUE;
		tyP0931MagConv2.tyDC.tyBtnSelClamp.uiMaskRtStat.0		:= TRUE;
		tyP0931MagConv2.tyDC.tyBtnSelUnclamp.uiMaskRtStat.0		:= TRUE;

		tyP0931MagConv2.tyCom.tyBtnSwitch.uiMaskRtStat.0		:= TRUE;

	END_IF

	IF EDGEPOS(bManualMod = FALSE) THEN
		tyP0931MagConv2.tyCom.tyBtnSwitch.bValue := FALSE;

		IF p_tyNtParamCurr.bMagAutoVerifyPrep = FALSE THEN
			fUIInRtStatHide(ADR(tyP0931MagConv2.tyDC.tyLyrWithoutSelClamp.uiRtStat));
			fUIInRtStatOff(ADR(tyP0931MagConv2.tyFB.tyLyrWithoutSelClamp.uiRtStat));
		ELSE

			fUIInRtStatHide(ADR(tyP0931MagConv2.tyDC.tyLyr.uiRtStat));
			fUIInRtStatOff(ADR(tyP0931MagConv2.tyFB.tyLyr.uiRtStat));
		END_IF
	END_IF
END_ACTION
```

#### Act_EntP0932Disp.st
```iecst
ACTION Act_EntP0932Disp:

	//Access Address
	p_tyC0002FullMask ACCESS ADR(tyP0932MagConv3.tyFullMaskHide);

//	p_tyC0004Navi ACCESS ADR(tyP0932MagConv3.tyNaviBack);

	p_tyC0004Navi ACCESS ADR(tyP0932MagConv3.tyNavi3Lyr3);

	p_tyC0005Main ACCESS ADR(tyCommon.tyMain);

	p_tyC0007Notif ACCESS ADR(tyCommon.tyNotif);

	p_tyC0008MsgBox ACCESS ADR(tyP0932MagConv3.tyMsgBoxHide);

	p_tyC0009Info ACCESS ADR(tyCommon.tyInfo);

	p_tyP0932Mag3ConvCom ACCESS ADR(tyP0932MagConv3.tyCom);
	p_tyP0932Mag3ConvDC ACCESS ADR(tyP0932MagConv3.tyDC);
	p_tyP0932Mag3ConvFB ACCESS ADR(tyP0932MagConv3.tyFB);

	tyP0931MagConv2.tyCom.tyBitmapMc.uiValueIdx	:= 235;

	IF p_tyNtParamCurr.bMagAutoVerifyPrep = FALSE THEN
		IF tyP0932MagConv3.tyCom.tyBtnSwitch.bValue THEN
			fUIInRtStatHide(ADR(tyP0932MagConv3.tyFB.tyLyr.uiRtStat));
			fUIInRtStatHide(ADR(tyP0932MagConv3.tyDC.tyLyr.uiRtStat));
			fUIInRtStatHide(ADR(tyP0932MagConv3.tyFB.tyLyrWithoutSelClamp.uiRtStat));
			fUIInRtStatOff(ADR(tyP0932MagConv3.tyDC.tyLyrWithoutSelClamp.uiRtStat));
		ELSE
			fUIInRtStatHide(ADR(tyP0932MagConv3.tyFB.tyLyr.uiRtStat));
			fUIInRtStatHide(ADR(tyP0932MagConv3.tyDC.tyLyr.uiRtStat));
			fUIInRtStatOff(ADR(tyP0932MagConv3.tyFB.tyLyrWithoutSelClamp.uiRtStat));
			fUIInRtStatHide(ADR(tyP0932MagConv3.tyDC.tyLyrWithoutSelClamp.uiRtStat));
		END_IF
	ELSE
		IF tyP0932MagConv3.tyCom.tyBtnSwitch.bValue THEN
			fUIInRtStatHide(ADR(tyP0932MagConv3.tyFB.tyLyr.uiRtStat));
			fUIInRtStatOff(ADR(tyP0932MagConv3.tyDC.tyLyr.uiRtStat));
			fUIInRtStatHide(ADR(tyP0932MagConv3.tyFB.tyLyrWithoutSelClamp.uiRtStat));
			fUIInRtStatHide(ADR(tyP0932MagConv3.tyDC.tyLyrWithoutSelClamp.uiRtStat));
		ELSE
			fUIInRtStatOff(ADR(tyP0932MagConv3.tyFB.tyLyr.uiRtStat));
			fUIInRtStatHide(ADR(tyP0932MagConv3.tyDC.tyLyr.uiRtStat));
			fUIInRtStatHide(ADR(tyP0932MagConv3.tyFB.tyLyrWithoutSelClamp.uiRtStat));
			fUIInRtStatHide(ADR(tyP0932MagConv3.tyDC.tyLyrWithoutSelClamp.uiRtStat));
		END_IF
	END_IF

END_ACTION
```

#### Act_OptP0932FullMask.st
```iecst
ACTION Act_OptP0932FullMask:

	IF eCurrPage = UIP0932MagConv3 THEN

		IF p_tyDI.bEStopSig = FALSE THEN
			p_tyC0002FullMask ACCESS ADR(tyP0932MagConv3.tyFullMaskEStop);

		ELSIF p_tyDI.bCoverSWSig = FALSE THEN
			p_tyC0002FullMask ACCESS ADR(tyP0932MagConv3.tyFullMaskCWSig);

		ELSIF p_tyDI.bSafetyRlySig = FALSE THEN
			p_tyC0002FullMask ACCESS ADR(tyP0932MagConv3.tyFullMaskSafetyRly);

		ELSIF p_bMag3AWEngageExtCtrl
			AND NOT p_bMagConv2Clp3ClprFixClampCtrl
			AND NOT p_bMagConv2Clp3ClprRmtClampCtrl
			THEN
			p_tyC0002FullMask ACCESS ADR(tyP0932MagConv3.tyFullMaskAWMotorEngage);

		ELSE
			p_tyC0002FullMask ACCESS ADR(tyP0932MagConv3.tyFullMaskHide);

		END_IF

	END_IF

END_ACTION
```

#### Act_OptP0932Navi.st
```iecst
ACTION Act_OptP0932Navi:

//	IF tyP0932MagConv3.tyNaviBack.tyBtnBack.bRtCompl = TRUE THEN
//		tyP0932MagConv3.tyNaviBack.tyBtnBack.bRtCompl	:= FALSE;
//		tyP0932MagConv3.tyNaviBack.tyBtnBack.bValue		:= FALSE;
//
//		eChgPage	:= UIP0920MtrNPneuCtrl;
//	END_IF

	IF tyP0932MagConv3.tyNavi3Lyr3.tyBtnBack.bRtCompl = TRUE THEN
		tyP0932MagConv3.tyNavi3Lyr3.tyBtnBack.bRtCompl	:= FALSE;
		tyP0932MagConv3.tyNavi3Lyr3.tyBtnBack.bValue		:= FALSE;

		eChgPage	:= UIP0920MtrNPneuCtrl;
		bDispMagConv1	:= FALSE;
		bDispMagConv2	:= FALSE;
		bDispMagConv3	:= TRUE;

	ELSIF tyP0932MagConv3.tyNavi3Lyr3.tyBtnLeft.bRtCompl = TRUE THEN
		tyP0932MagConv3.tyNavi3Lyr3.tyBtnLeft.bRtCompl				:= FALSE;
		tyP0932MagConv3.tyNavi3Lyr3.tyBtnLeft.bValue				:= FALSE;
		eChgPage													:= UIP0931MagConv2;
		bDispMagConv1	:= FALSE;
		bDispMagConv2	:= TRUE;
		bDispMagConv3	:= FALSE;

	ELSIF tyP0932MagConv3.tyNavi3Lyr3.tyBtnRgt.bRtCompl = TRUE THEN
			tyP0932MagConv3.tyNavi3Lyr3.tyBtnRgt.bRtCompl			:= FALSE;
			tyP0932MagConv3.tyNavi3Lyr3.tyBtnRgt.bValue				:= FALSE;
			eChgPage												:= UIP0930MagConv1;
			bDispMagConv1	:= FALSE;
			bDispMagConv2	:= FALSE;
			bDispMagConv3	:= TRUE;
	END_IF

END_ACTION
```

#### Act_OptP0932MagConv3ChgLyr.st
```iecst
ACTION Act_OptP0932MagConv3ChgLyr:

	IF p_tyNtParamCurr.bMagAutoVerifyPrep THEN
		IF tyP0932MagConv3.tyCom.tyBtnSwitch.bRtCompl THEN
			tyP0932MagConv3.tyCom.tyBtnSwitch.bRtCompl := FALSE;

			IF tyP0932MagConv3.tyCom.tyBtnSwitch.bValue = TRUE THEN
				fUIInRtStatOff(ADR(tyP0932MagConv3.tyDC.tyLyr.uiRtStat));
				fUIInRtStatHide(ADR(tyP0932MagConv3.tyFB.tyLyr.uiRtStat));
			ELSE
				fUIInRtStatHide(ADR(tyP0932MagConv3.tyDC.tyLyr.uiRtStat));
				fUIInRtStatOff(ADR(tyP0932MagConv3.tyFB.tyLyr.uiRtStat));
			END_IF

		END_IF
	ELSE
		IF tyP0932MagConv3.tyCom.tyBtnSwitch.bRtCompl THEN
			tyP0932MagConv3.tyCom.tyBtnSwitch.bRtCompl	:= FALSE;

			IF tyP0932MagConv3.tyCom.tyBtnSwitch.bValue = TRUE THEN
				fUIInRtStatOff(ADR(tyP0932MagConv3.tyDC.tyLyrWithoutSelClamp.uiRtStat));
				fUIInRtStatHide(ADR(tyP0932MagConv3.tyFB.tyLyrWithoutSelClamp.uiRtStat));
			ELSE
				fUIInRtStatHide(ADR(tyP0932MagConv3.tyDC.tyLyrWithoutSelClamp.uiRtStat));
				fUIInRtStatOff(ADR(tyP0932MagConv3.tyFB.tyLyrWithoutSelClamp.uiRtStat));
			END_IF

		END_IF
	END_IF

END_ACTION
```

#### Act_OptP0932MagConv3Sen.st
```iecst
ACTION Act_OptP0932MagConv3Sen:

	tyP0932MagConv3.tyCom.tyBtnMagPresentSen.bValue			:= p_tyDI.bMagPresentSen3;
	tyP0932MagConv3.tyCom.tyBtnMagConvEntSen.bValue			:= p_tyDI.bMagConvEntSen3;
	tyP0932MagConv3.tyCom.tyBtnMagAIVPosSen1.bValue			:= p_tyDI.bMag3AIVInPosSen1;
	tyP0932MagConv3.tyCom.tyBtnMagAIVPosSen2.bValue			:= p_tyDI.bMag3AIVInPosSen2;
	tyP0932MagConv3.tyCom.tyBtnMagOrientationChkSen1.bValue	:= p_tyDI.bMag3OrientChkSen1;
	tyP0932MagConv3.tyCom.tyBtnMagOrientationChkSen2.bValue	:= p_tyDI.bMag3OrientChkSen2;

	tyP0932MagConv3.tyCom.tyBtnFixedClampRS.bValue			:= p_tyDI.bMag3FixedClampRS;
	tyP0932MagConv3.tyCom.tyBtnFixedUnclampRS.bValue		:= p_tyDI.bMag3FixedUnclampRS;
	tyP0932MagConv3.tyCom.tyBtnRemoteClampRS.bValue			:= p_tyDI.bMag3RemoteClampRS;
	tyP0932MagConv3.tyCom.tyBtnRemoteUnclampRS.bValue		:= p_tyDI.bMag3RemoteUnclampRS;

	tyP0932MagConv3.tyCom.tyBtnSelUnclampRS.bValue			:= p_tyDI.bMag3SelUnClampRS;

	tyP0932MagConv3.tyCom.tyBtnCAB717Sen.bValue				:= p_tyDI.bMagConvCAB717MagSen3;
//	tyP0932MagConv3.tyCom.tyBtnHeightSen.bValue				:= p_tyDI.bMagConvHeightSen3;
	tyP0932MagConv3.tyCom.tyBtnMagSmallSen.bValue			:= p_tyDI.bMagConvSmallMagSen3;
	tyP0932MagConv3.tyCom.tyBtnMagLargeSen.bValue			:= p_tyDI.bMagConvLargeMagSen3;

	tyP0932MagConv3.tyCom.tyBtnMagDetectSen.bValue			:= p_tyDI.bMag3FixedClampSen;
//	tyP0932MagConv3.tyCom.tyBtnMagDetectSen.uiRtStat.0		:= NOT p_tyNtParamCurr.bProjFixClprMagDetectSenPrep;

	IF p_tyNtParamCurr.bMagAutoVerifyPrep = TRUE THEN
		tyP0932MagConv3.tyCom.tyBtnHeightSen.bValue			:= p_tyDI.bMagConvHeightSen3;
	ELSE
		tyP0932MagConv3.tyCom.tyBtnHeightSen.bValue			:= p_tyDI.bHighMagDetSen3;
	END_IF

	//Machine Bitmap
	IF p_tyNtParamCurr.bMagAutoVerifyPrep = FALSE AND p_tyNtParamCurr.bProjMotorizedPusherPrep = FALSE THEN
	IF tyP0932MagConv3.tyFB.tyBtnFixedClamp.bRtCompl OR  tyP0932MagConv3.tyFB.tyBtnRemoteClamp.bRtCompl
		OR tyP0932MagConv3.tyDC.tyBtnFixedClamp.bRtCompl OR tyP0932MagConv3.tyDC.tyBtnRemoteClamp.bRtCompl  THEN

		tyP0932MagConv3.tyCom.tyBitmapMc.uiValueIdx	:= 2;

	ELSIF tyP0932MagConv3.tyFB.tyBtnFixedUnclamp.bRtCompl OR tyP0932MagConv3.tyFB.tyBtnRemoteUnclamp.bRtCompl
		OR tyP0932MagConv3.tyDC.tyBtnFixedUnclamp.bRtCompl OR tyP0932MagConv3.tyDC.tyBtnRemoteUnclamp.bRtCompl  THEN

		tyP0932MagConv3.tyCom.tyBitmapMc.uiValueIdx	:= 1;

	ELSIF tyP0932MagConv3.tyFB.tyBtnEnt.bRtCompl OR tyP0932MagConv3.tyFB.tyBtnExit.bRtCompl OR tyP0932MagConv3.tyFB.tyBtnStop.bRtCompl
		OR tyP0932MagConv3.tyDC.tyBtnMagIn.bRtCompl OR tyP0932MagConv3.tyDC.tyBtnMagOut.bRtCompl OR tyP0932MagConv3.tyDC.tyBtnStop.bRtCompl THEN

		tyP0932MagConv3.tyCom.tyBitmapMc.uiValueIdx	:= 0;

	END_IF
ELSIF p_tyNtParamCurr.bMagAutoVerifyPrep AND p_tyNtParamCurr.bProjMagAWPrep = FALSE AND p_tyNtParamCurr.bProjMotorizedPusherPrep = FALSE THEN
		IF tyP0932MagConv3.tyFB.tyBtnFixedClamp.bRtCompl (*Bottom*)
			OR tyP0932MagConv3.tyDC.tyBtnFixedClamp.bRtCompl THEN

			tyP0932MagConv3.tyCom.tyBitmapMc.uiValueIdx	:= 24;

		ELSIF tyP0932MagConv3.tyFB.tyBtnFixedUnclamp.bRtCompl
			OR tyP0932MagConv3.tyDC.tyBtnFixedUnclamp.bRtCompl THEN

			tyP0932MagConv3.tyCom.tyBitmapMc.uiValueIdx	:= 25;

		ELSIF tyP0932MagConv3.tyFB.tyBtnRemoteClamp.bRtCompl (*Top*)
			OR tyP0932MagConv3.tyDC.tyBtnRemoteClamp.bRtCompl THEN

			tyP0932MagConv3.tyCom.tyBitmapMc.uiValueIdx	:= 19;

		ELSIF tyP0932MagConv3.tyFB.tyBtnRemoteUnclamp.bRtCompl
			OR tyP0932MagConv3.tyDC.tyBtnRemoteUnclamp.bRtCompl THEN

			tyP0932MagConv3.tyCom.tyBitmapMc.uiValueIdx	:= 18;

		ELSIF tyP0932MagConv3.tyFB.tyBtnSelClamp.bRtCompl
			OR tyP0932MagConv3.tyDC.tyBtnSelClamp.bRtCompl THEN

			tyP0932MagConv3.tyCom.tyBitmapMc.uiValueIdx	:= 31;

		ELSIF tyP0932MagConv3.tyFB.tyBtnSelUnclamp.bRtCompl
			OR tyP0932MagConv3.tyDC.tyBtnSelUnclamp.bRtCompl THEN

			tyP0932MagConv3.tyCom.tyBitmapMc.uiValueIdx	:= 30;

		ELSIF tyP0932MagConv3.tyFB.tyBtnEnt.bRtCompl OR tyP0932MagConv3.tyFB.tyBtnExit.bRtCompl OR tyP0932MagConv3.tyFB.tyBtnStop.bRtCompl
			OR tyP0932MagConv3.tyDC.tyBtnMagIn.bRtCompl OR tyP0932MagConv3.tyDC.tyBtnMagOut.bRtCompl OR tyP0932MagConv3.tyDC.tyBtnStop.bRtCompl THEN

			tyP0932MagConv3.tyCom.tyBitmapMc.uiValueIdx	:= 0;

		END_IF

	ELSIF p_tyNtParamCurr.bMagAutoVerifyPrep AND p_tyNtParamCurr.bProjMagAWPrep THEN
		IF tyP0932MagConv3.tyFB.tyBtnFixedClamp.bRtCompl (*Bottom*)
			OR tyP0932MagConv3.tyDC.tyBtnFixedClamp.bRtCompl THEN

			tyP0932MagConv3.tyCom.tyBitmapMc.uiValueIdx	:= 48;

		ELSIF tyP0932MagConv3.tyFB.tyBtnFixedUnclamp.bRtCompl
			OR tyP0932MagConv3.tyDC.tyBtnFixedUnclamp.bRtCompl THEN

			tyP0932MagConv3.tyCom.tyBitmapMc.uiValueIdx	:= 49;

		ELSIF tyP0932MagConv3.tyFB.tyBtnRemoteClamp.bRtCompl (*Top*)
			OR tyP0932MagConv3.tyDC.tyBtnRemoteClamp.bRtCompl THEN

			tyP0932MagConv3.tyCom.tyBitmapMc.uiValueIdx	:= 61;

		ELSIF tyP0932MagConv3.tyFB.tyBtnRemoteUnclamp.bRtCompl
			OR tyP0932MagConv3.tyDC.tyBtnRemoteUnclamp.bRtCompl THEN

			tyP0932MagConv3.tyCom.tyBitmapMc.uiValueIdx	:= 60;

		ELSIF tyP0932MagConv3.tyFB.tyBtnSelClamp.bRtCompl
			OR tyP0932MagConv3.tyDC.tyBtnSelClamp.bRtCompl THEN

			tyP0932MagConv3.tyCom.tyBitmapMc.uiValueIdx	:= 43;

		ELSIF tyP0932MagConv3.tyFB.tyBtnSelUnclamp.bRtCompl
			OR tyP0932MagConv3.tyDC.tyBtnSelUnclamp.bRtCompl THEN

			tyP0932MagConv3.tyCom.tyBitmapMc.uiValueIdx	:= 42;

		ELSIF tyP0932MagConv3.tyFB.tyBtnEnt.bRtCompl OR tyP0932MagConv3.tyFB.tyBtnExit.bRtCompl OR tyP0932MagConv3.tyFB.tyBtnStop.bRtCompl
			OR tyP0932MagConv3.tyDC.tyBtnMagIn.bRtCompl OR tyP0932MagConv3.tyDC.tyBtnMagOut.bRtCompl OR tyP0932MagConv3.tyDC.tyBtnStop.bRtCompl THEN

			tyP0932MagConv3.tyCom.tyBitmapMc.uiValueIdx	:= 3;

		END_IF

	ELSIF p_tyNtParamCurr.bMagAutoVerifyPrep = FALSE AND p_tyNtParamCurr.bProjMagAWPrep = FALSE AND p_tyNtParamCurr.bProjMotorizedPusherPrep THEN
		IF tyP0932MagConv3.tyFB.tyBtnFixedClamp.bRtCompl
			OR tyP0932MagConv3.tyDC.tyBtnFixedClamp.bRtCompl THEN

			IF p_tyNtParamCurr.bCurtainSenPrep THEN
				tyP0932MagConv3.tyCom.tyBitmapMc.uiValueIdx	:= 234;
			ELSE
				tyP0932MagConv3.tyCom.tyBitmapMc.uiValueIdx	:= 207;
			END_IF

		ELSIF tyP0932MagConv3.tyFB.tyBtnFixedUnclamp.bRtCompl
			OR tyP0932MagConv3.tyDC.tyBtnFixedUnclamp.bRtCompl THEN

			IF p_tyNtParamCurr.bCurtainSenPrep THEN
				tyP0932MagConv3.tyCom.tyBitmapMc.uiValueIdx	:= 234;
			ELSE
				tyP0932MagConv3.tyCom.tyBitmapMc.uiValueIdx	:= 206;
			END_IF

		ELSIF tyP0932MagConv3.tyFB.tyBtnRemoteClamp.bRtCompl
			OR tyP0932MagConv3.tyDC.tyBtnRemoteClamp.bRtCompl THEN

			IF p_tyNtParamCurr.bCurtainSenPrep THEN
				tyP0932MagConv3.tyCom.tyBitmapMc.uiValueIdx	:= 234;
			ELSE
				tyP0932MagConv3.tyCom.tyBitmapMc.uiValueIdx	:= 219;
			END_IF

		ELSIF tyP0932MagConv3.tyFB.tyBtnRemoteUnclamp.bRtCompl
			OR tyP0932MagConv3.tyDC.tyBtnRemoteUnclamp.bRtCompl THEN

			IF p_tyNtParamCurr.bCurtainSenPrep THEN
				tyP0932MagConv3.tyCom.tyBitmapMc.uiValueIdx	:= 234;
			ELSE
				tyP0932MagConv3.tyCom.tyBitmapMc.uiValueIdx	:= 218;
			END_IF

			//				ELSIF tyP0930MagConv3.tyFB.tyBtnSelClamp.bRtCompl
			//					OR tyP0930MagConv3.tyDC.tyBtnSelClamp.bRtCompl THEN
			//
			//					tyP0930MagConv3.tyCom.tyBitmapMc.uiValueIdx	:= 41;
			//
			//				ELSIF tyP0930MagConv3.tyFB.tyBtnSelUnclamp.bRtCompl
			//					OR tyP0930MagConv3.tyDC.tyBtnSelUnclamp.bRtCompl THEN
			//
			//					tyP0930MagConv3.tyCom.tyBitmapMc.uiValueIdx	:= 40;
			//
		ELSIF tyP0932MagConv3.tyFB.tyBtnEnt.bRtCompl OR tyP0932MagConv3.tyFB.tyBtnExit.bRtCompl OR tyP0932MagConv3.tyFB.tyBtnStop.bRtCompl
			OR tyP0932MagConv3.tyDC.tyBtnMagIn.bRtCompl OR tyP0932MagConv3.tyDC.tyBtnMagOut.bRtCompl OR tyP0932MagConv3.tyDC.tyBtnStop.bRtCompl THEN

			IF p_tyNtParamCurr.bCurtainSenPrep THEN
				tyP0932MagConv3.tyCom.tyBitmapMc.uiValueIdx	:= 235;
			ELSE
				tyP0932MagConv3.tyCom.tyBitmapMc.uiValueIdx	:= 205;
			END_IF

		END_IF
	END_IF

//	IF p_tyNtParamCurr.eProjMag = ULMagTriple AND p_tyNtParamCurr.bMagAutoVerifyPrep = FALSE THEN
//		IF tyP0932MagConv3.tyCom.tyBitmapMc.uiValueIdx < 100 THEN
//			tyP0932MagConv3.tyCom.tyBitmapMc.uiValueIdx	:= tyP0932MagConv3.tyCom.tyBitmapMc.uiValueIdx + 100;
//		END_IF
//	ELSIF p_tyNtParamCurr.eProjMag = ULMagTriple AND p_tyNtParamCurr.bMagAutoVerifyPrep = TRUE THEN
//		IF tyP0932MagConv3.tyCom.tyBitmapMc.uiValueIdx < 200 THEN
//			tyP0932MagConv3.tyCom.tyBitmapMc.uiValueIdx	:= tyP0932MagConv3.tyCom.tyBitmapMc.uiValueIdx + 200;
//		END_IF
//	END_IF

END_ACTION
```

#### Act_OptP0932MagConv3FB.st
```iecst
ACTION Act_OptP0932MagConv3FB:

	//Magazine Conveyor
	IF tyP0932MagConv3.tyFB.tyBtnStop.bRtCompl = TRUE THEN
		eMagConv2Clp3Act	:= MagConv2ClpActStop;

		IF p_eMagConv2Clp3Stat = MagConv2ClpActStop AND p_eMagConv2Clp3Status = Done THEN
			eMagConv2Clp3Act	:= MagConv2ClpActIdle;

			tyP0932MagConv3.tyFB.tyBtnEnt.bRtCompl	:= FALSE;
			tyP0932MagConv3.tyFB.tyBtnEnt.bValue	:= FALSE;
			tyP0932MagConv3.tyFB.tyBtnEnt.bRtLk		:= FALSE;

			tyP0932MagConv3.tyFB.tyBtnExit.bRtCompl	:= FALSE;
			tyP0932MagConv3.tyFB.tyBtnExit.bValue	:= FALSE;
			tyP0932MagConv3.tyFB.tyBtnExit.bRtLk	:= FALSE;

			tyP0932MagConv3.tyFB.tyBtnStop.bRtCompl	:= FALSE;
			tyP0932MagConv3.tyFB.tyBtnStop.bValue	:= TRUE;
			tyP0932MagConv3.tyFB.tyBtnStop.bRtLk	:= TRUE;
		END_IF

	ELSIF tyP0932MagConv3.tyFB.tyBtnEnt.bRtCompl = TRUE THEN
		tyP0932MagConv3.tyFB.tyBtnEnt.bValue	:= TRUE;
		tyP0932MagConv3.tyFB.tyBtnEnt.bRtLk		:= TRUE;

		tyP0932MagConv3.tyFB.tyBtnStop.bValue	:= FALSE;
		tyP0932MagConv3.tyFB.tyBtnStop.bRtLk	:= FALSE;

		eMagConv2Clp3Act	:= MagConv2ClpActEnt;

		IF p_eMagConv2Clp3Stat = MagConv2ClpActEnt AND p_eMagConv2Clp3Status = Done THEN
			eMagConv2Clp3Act	:= MagConv2ClpActIdle;

			tyP0932MagConv3.tyFB.tyBtnEnt.bRtCompl	:= FALSE;

			tyP0932MagConv3.tyFB.tyBtnEnt.bValue	:= FALSE;
			tyP0932MagConv3.tyFB.tyBtnEnt.bRtLk		:= FALSE;

			tyP0932MagConv3.tyFB.tyBtnStop.bValue	:= TRUE;
			tyP0932MagConv3.tyFB.tyBtnStop.bRtLk	:= TRUE;
		END_IF

	ELSIF (p_eMagConv2Clp3Stat = MagConv2ClpActPreExit AND p_eMagConv2Clp3Status = Done) THEN
		eMagConv2Clp3Act	:= MagConv2ClpActIdle;

		tyP0932MagConv3.tyFB.tyBtnExit.bRtCompl	:= FALSE;

		tyP0932MagConv3.tyFB.tyBtnExit.bValue	:= FALSE;
		tyP0932MagConv3.tyFB.tyBtnExit.bRtLk	:= FALSE;

		tyP0932MagConv3.tyFB.tyBtnStop.bValue	:= TRUE;
		tyP0932MagConv3.tyFB.tyBtnStop.bRtLk	:= TRUE;

	ELSIF (p_eMagConv2Clp3Stat = MagConv2ClpActExit AND p_eMagConv2Clp3Status = Done) THEN
		eMagConv2Clp3Act	:= MagConv2ClpActIdle;

		tyP0932MagConv3.tyFB.tyBtnExit.bRtCompl	:= FALSE;

		tyP0932MagConv3.tyFB.tyBtnExit.bValue	:= FALSE;
		tyP0932MagConv3.tyFB.tyBtnExit.bRtLk	:= FALSE;

		tyP0932MagConv3.tyFB.tyBtnStop.bValue	:= TRUE;
		tyP0932MagConv3.tyFB.tyBtnStop.bRtLk	:= TRUE;

	ELSIF tyP0932MagConv3.tyFB.tyBtnExit.bRtCompl = TRUE THEN
		tyP0932MagConv3.tyFB.tyBtnExit.bRtCompl	:= FALSE;
		tyP0932MagConv3.tyFB.tyBtnExit.bValue	:= TRUE;
		tyP0932MagConv3.tyFB.tyBtnExit.bRtLk	:= TRUE;

		tyP0932MagConv3.tyFB.tyBtnStop.bValue	:= FALSE;
		tyP0932MagConv3.tyFB.tyBtnStop.bRtLk	:= FALSE;

		IF p_tyDI.bMagConvEntSen3  THEN
			eMagConv2Clp3Act	:= MagConv2ClpActExit;
		ELSE
			IF p_tyDI.bMagPresentSen3 THEN
				eMagConv2Clp3Act	:= MagConv2ClpActPreExit;
			ELSE
				eMagConv2Clp3Act	:= MagConv2ClpActExit;
			END_IF
		END_IF
	END_IF

	//Magazine Clamper
	IF tyP0932MagConv3.tyCom.tyBtnSwitch.bValue = FALSE THEN

		//Fixed
		IF tyP0932MagConv3.tyFB.tyBtnFixedUnclamp.bRtCompl = TRUE THEN
			tyP0932MagConv3.tyFB.tyBtnFixedUnclamp.bRtCompl	:= FALSE;

			tyP0932MagConv3.tyFB.tyBtnFixedUnclamp.bValue	:= TRUE;
			tyP0932MagConv3.tyFB.tyBtnFixedClamp.bValue		:= FALSE;

		ELSIF tyP0932MagConv3.tyFB.tyBtnFixedClamp.bRtCompl = TRUE THEN
			tyP0932MagConv3.tyFB.tyBtnFixedClamp.bRtCompl	:= FALSE;

			tyP0932MagConv3.tyFB.tyBtnFixedClamp.bValue		:= TRUE;
			tyP0932MagConv3.tyFB.tyBtnFixedUnclamp.bValue	:= FALSE;

		END_IF

		//Remote
		IF tyP0932MagConv3.tyFB.tyBtnRemoteUnclamp.bRtCompl = TRUE THEN
			tyP0932MagConv3.tyFB.tyBtnRemoteUnclamp.bRtCompl	:= FALSE;

			tyP0932MagConv3.tyFB.tyBtnRemoteUnclamp.bValue	:= TRUE;
			tyP0932MagConv3.tyFB.tyBtnRemoteClamp.bValue	:= FALSE;

		ELSIF tyP0932MagConv3.tyFB.tyBtnRemoteClamp.bRtCompl = TRUE THEN
			tyP0932MagConv3.tyFB.tyBtnRemoteClamp.bRtCompl	:= FALSE;

			tyP0932MagConv3.tyFB.tyBtnRemoteClamp.bValue	:= TRUE;
			tyP0932MagConv3.tyFB.tyBtnRemoteUnclamp.bValue	:= FALSE;

		END_IF

		//Selection
		IF tyP0932MagConv3.tyFB.tyBtnSelUnclamp.bRtCompl = TRUE THEN
			tyP0932MagConv3.tyFB.tyBtnSelUnclamp.bRtCompl	:= FALSE;

			tyP0932MagConv3.tyFB.tyBtnSelUnclamp.bValue	:= TRUE;
			tyP0932MagConv3.tyFB.tyBtnSelClamp.bValue	:= FALSE;

		ELSIF tyP0932MagConv3.tyFB.tyBtnSelClamp.bRtCompl = TRUE THEN
			tyP0932MagConv3.tyFB.tyBtnSelClamp.bRtCompl	:= FALSE;

			tyP0932MagConv3.tyFB.tyBtnSelClamp.bValue	:= TRUE;
			tyP0932MagConv3.tyFB.tyBtnSelUnclamp.bValue	:= FALSE;

		END_IF

		// Fixed Clamper
		IF tyP0932MagConv3.tyFB.tyBtnFixedUnclamp.bValue = TRUE THEN

			eMagConv2Clp3Act	:= MagConv2ClpActFixClprUnclamp;

			IF p_eMagConv2Clp3Stat = MagConv2ClpActFixClprUnclamp AND p_eMagConv2Clp3Status = Done THEN

				eMagConv2Clp3Act	:= MagConv2ClpActIdle;

				tyP0932MagConv3.tyFB.tyBtnFixedUnclamp.bValue	:= FALSE;

			ELSIF p_eMagConv2Clp3Status = Error THEN

				tyP0932MagConv3.tyFB.tyBtnFixedUnclamp.bValue	:= FALSE;

			END_IF

		ELSIF tyP0932MagConv3.tyFB.tyBtnFixedClamp.bValue = TRUE THEN
			eMagConv2Clp3Act	:= MagConv2ClpActFixClprClamp;

			IF p_eMagConv2Clp3Stat = MagConv2ClpActFixClprClamp AND p_eMagConv2Clp3Status = Done THEN

				eMagConv2Clp3Act	:= MagConv2ClpActIdle;

				tyP0932MagConv3.tyFB.tyBtnFixedClamp.bValue := FALSE;

			ELSIF p_eMagConv2Clp3Status = Error THEN
				tyP0932MagConv3.tyFB.tyBtnFixedClamp.bValue := FALSE;

			END_IF

			//Sel
			IF tyP0932MagConv3.tyFB.tyBtnSelUnclamp.bRtCompl = TRUE THEN
				tyP0932MagConv3.tyFB.tyBtnSelUnclamp.bRtCompl	:= FALSE;

				tyP0932MagConv3.tyFB.tyBtnSelUnclamp.bValue	:= TRUE;
				tyP0932MagConv3.tyFB.tyBtnSelClamp.bValue	:= FALSE;

			ELSIF tyP0932MagConv3.tyFB.tyBtnSelClamp.bRtCompl = TRUE THEN
				tyP0932MagConv3.tyFB.tyBtnSelClamp.bRtCompl	:= FALSE;

				tyP0932MagConv3.tyFB.tyBtnSelClamp.bValue	:= TRUE;
				tyP0932MagConv3.tyFB.tyBtnSelUnclamp.bValue	:= FALSE;

			END_IF

		END_IF

		//Remote Clamper
		IF tyP0932MagConv3.tyFB.tyBtnRemoteUnclamp.bValue = TRUE THEN

			eMagConv2Clp3Act	:= MagConv2ClpActRmtClprUnclamp;

			IF p_eMagConv2Clp3Stat = MagConv2ClpActRmtClprUnclamp AND p_eMagConv2Clp3Status = Done THEN

				eMagConv2Clp3Act	:= MagConv2ClpActIdle;

				tyP0932MagConv3.tyFB.tyBtnRemoteUnclamp.bValue	:= FALSE;

			ELSIF p_eMagConv2Clp3Status = Error THEN

				tyP0932MagConv3.tyFB.tyBtnRemoteUnclamp.bValue	:= FALSE;

			END_IF

		ELSIF tyP0932MagConv3.tyFB.tyBtnRemoteClamp.bValue = TRUE THEN
			eMagConv2Clp3Act	:= MagConv2ClpActRmtClprClamp;

			IF p_eMagConv2Clp3Stat = MagConv2ClpActRmtClprClamp AND p_eMagConv2Clp3Status = Done THEN

				eMagConv2Clp3Act	:= MagConv2ClpActIdle;

				tyP0932MagConv3.tyFB.tyBtnRemoteClamp.bValue := FALSE;

			ELSIF p_eMagConv2Clp3Status = Error THEN
				tyP0932MagConv3.tyFB.tyBtnRemoteClamp.bValue := FALSE;

			END_IF

		END_IF

		//Selection Clamper
		IF tyP0932MagConv3.tyFB.tyBtnSelUnclamp.bValue = TRUE THEN

			eMagConvSelClp3Act	:= PneuActExt;

			IF p_eSelClamp3Stat = PneuActExt AND p_eSelClamp3Status = Done THEN

				eMagConvSelClp3Act	:= PneuActIdle;

				tyP0932MagConv3.tyFB.tyBtnSelUnclamp.bValue	:= FALSE;

			ELSIF p_eSelClamp3Status = Error THEN

				tyP0932MagConv3.tyFB.tyBtnSelUnclamp.bValue	:= FALSE;

			END_IF

		ELSIF tyP0932MagConv3.tyFB.tyBtnSelClamp.bValue = TRUE THEN
			eMagConvSelClp3Act	:= PneuActRet;

			IF p_eSelClamp3Stat = PneuActRet AND p_eSelClamp3Status = Done THEN

				eMagConvSelClp3Act	:= PneuActIdle;

				tyP0932MagConv3.tyFB.tyBtnSelClamp.bValue	:= FALSE;

			ELSIF p_eSelClamp3Status = Error THEN
				tyP0932MagConv3.tyFB.tyBtnSelClamp.bValue	:= FALSE;

			END_IF

		END_IF

		//Update Status
		tyP0932MagConv3.tyDC.tyBtnFixedUnclamp.bValue	:= NOT p_bMagConv2Clp3ClprFixClampCtrl;
		tyP0932MagConv3.tyDC.tyBtnFixedClamp.bValue		:= p_bMagConv2Clp3ClprFixClampCtrl;
		tyP0932MagConv3.tyDC.tyBtnRemoteUnclamp.bValue	:= NOT p_bMagConv2Clp3ClprRmtClampCtrl;
		tyP0932MagConv3.tyDC.tyBtnRemoteClamp.bValue	:= p_bMagConv2Clp3ClprRmtClampCtrl;

		tyP0932MagConv3.tyDC.tyBtnSelUnclamp.bRtCompl	:= FALSE;
		tyP0932MagConv3.tyDC.tyBtnSelClamp.bRtCompl		:= FALSE;
		tyP0932MagConv3.tyDC.tyBtnSelUnclamp.bValue	:= p_bSelClamp3RetCtrl;
		tyP0932MagConv3.tyDC.tyBtnSelClamp.bValue	:= p_bSelClamp3ExtCtrl;
	END_IF

	//Mask
	IF p_tyUsrMgmtCurrAccessRgt.bManualFBOnly THEN

		fUIInRtStatOff(ADR(tyP0932MagConv3.tyCom.tyBtnSwitch.uiMaskRtStat));

	ELSE

	IF p_eMagConv2Clp3Status = Error THEN

		fUIInRtStatOff(ADR(tyP0932MagConv3.tyFB.tyBtnEnt.uiMaskRtStat));
		fUIInRtStatOff(ADR(tyP0932MagConv3.tyFB.tyBtnExit.uiMaskRtStat));
		fUIInRtStatOff(ADR(tyP0932MagConv3.tyFB.tyBtnFixedClamp.uiMaskRtStat));
		fUIInRtStatOff(ADR(tyP0932MagConv3.tyFB.tyBtnFixedUnclamp.uiMaskRtStat));
		fUIInRtStatOff(ADR(tyP0932MagConv3.tyFB.tyBtnRemoteClamp.uiMaskRtStat));
		fUIInRtStatOff(ADR(tyP0932MagConv3.tyFB.tyBtnRemoteUnclamp.uiMaskRtStat));
			fUIInRtStatOff(ADR(tyP0932MagConv3.tyFB.tyBtnSelClamp.uiMaskRtStat));
			fUIInRtStatOff(ADR(tyP0932MagConv3.tyFB.tyBtnSelUnclamp.uiMaskRtStat));
		fUIInRtStatHide(ADR(tyP0932MagConv3.tyCom.tyBtnSwitch.uiMaskRtStat));

	ELSIF tyP0932MagConv3.tyFB.tyBtnEnt.bRtCompl = TRUE THEN

		fUIInRtStatHide(ADR(tyP0932MagConv3.tyFB.tyBtnEnt.uiMaskRtStat));
		fUIInRtStatOff(ADR(tyP0932MagConv3.tyFB.tyBtnExit.uiMaskRtStat));
		fUIInRtStatOff(ADR(tyP0932MagConv3.tyFB.tyBtnFixedClamp.uiMaskRtStat));
		fUIInRtStatOff(ADR(tyP0932MagConv3.tyFB.tyBtnFixedUnclamp.uiMaskRtStat));
		fUIInRtStatOff(ADR(tyP0932MagConv3.tyFB.tyBtnRemoteClamp.uiMaskRtStat));
		fUIInRtStatOff(ADR(tyP0932MagConv3.tyFB.tyBtnRemoteUnclamp.uiMaskRtStat));
			fUIInRtStatOff(ADR(tyP0932MagConv3.tyFB.tyBtnSelClamp.uiMaskRtStat));
			fUIInRtStatOff(ADR(tyP0932MagConv3.tyFB.tyBtnSelUnclamp.uiMaskRtStat));
		fUIInRtStatOff(ADR(tyP0932MagConv3.tyCom.tyBtnSwitch.uiMaskRtStat));

	ELSIF tyP0932MagConv3.tyFB.tyBtnExit.bRtCompl = TRUE THEN

		fUIInRtStatOff(ADR(tyP0932MagConv3.tyFB.tyBtnEnt.uiMaskRtStat));
		fUIInRtStatHide(ADR(tyP0932MagConv3.tyFB.tyBtnExit.uiMaskRtStat));
		fUIInRtStatOff(ADR(tyP0932MagConv3.tyFB.tyBtnFixedClamp.uiMaskRtStat));
		fUIInRtStatOff(ADR(tyP0932MagConv3.tyFB.tyBtnFixedUnclamp.uiMaskRtStat));
		fUIInRtStatOff(ADR(tyP0932MagConv3.tyFB.tyBtnRemoteClamp.uiMaskRtStat));
		fUIInRtStatOff(ADR(tyP0932MagConv3.tyFB.tyBtnRemoteUnclamp.uiMaskRtStat));
		fUIInRtStatOff(ADR(tyP0932MagConv3.tyFB.tyBtnSelClamp.uiMaskRtStat));
		fUIInRtStatOff(ADR(tyP0932MagConv3.tyFB.tyBtnSelUnclamp.uiMaskRtStat));
		fUIInRtStatOff(ADR(tyP0932MagConv3.tyCom.tyBtnSwitch.uiMaskRtStat));

	ELSIF tyP0932MagConv3.tyFB.tyBtnFixedClamp.bValue = TRUE OR tyP0932MagConv3.tyFB.tyBtnRemoteClamp.bValue = TRUE
			OR tyP0932MagConv3.tyFB.tyBtnFixedUnclamp.bValue = TRUE OR tyP0932MagConv3.tyFB.tyBtnRemoteUnclamp.bValue = TRUE
			OR tyP0932MagConv3.tyFB.tyBtnSelClamp.bValue = TRUE OR tyP0932MagConv3.tyFB.tyBtnSelUnclamp.bValue = TRUE
			THEN

		fUIInRtStatOff(ADR(tyP0932MagConv3.tyFB.tyBtnEnt.uiMaskRtStat));
		fUIInRtStatOff(ADR(tyP0932MagConv3.tyFB.tyBtnExit.uiMaskRtStat));
		fUIInRtStatHide(ADR(tyP0932MagConv3.tyFB.tyBtnFixedClamp.uiMaskRtStat));
		fUIInRtStatHide(ADR(tyP0932MagConv3.tyFB.tyBtnFixedUnclamp.uiMaskRtStat));
		fUIInRtStatHide(ADR(tyP0932MagConv3.tyFB.tyBtnRemoteClamp.uiMaskRtStat));
		fUIInRtStatHide(ADR(tyP0932MagConv3.tyFB.tyBtnRemoteUnclamp.uiMaskRtStat));
		fUIInRtStatHide(ADR(tyP0932MagConv3.tyFB.tyBtnSelClamp.uiMaskRtStat));
		fUIInRtStatHide(ADR(tyP0932MagConv3.tyFB.tyBtnSelUnclamp.uiMaskRtStat));
		fUIInRtStatOff(ADR(tyP0932MagConv3.tyCom.tyBtnSwitch.uiMaskRtStat));

	ELSE

		fUIInRtStatHide(ADR(tyP0932MagConv3.tyFB.tyBtnEnt.uiMaskRtStat));
		fUIInRtStatHide(ADR(tyP0932MagConv3.tyFB.tyBtnExit.uiMaskRtStat));
		fUIInRtStatHide(ADR(tyP0932MagConv3.tyFB.tyBtnFixedClamp.uiMaskRtStat));
		fUIInRtStatHide(ADR(tyP0932MagConv3.tyFB.tyBtnFixedUnclamp.uiMaskRtStat));
		fUIInRtStatHide(ADR(tyP0932MagConv3.tyFB.tyBtnRemoteClamp.uiMaskRtStat));
		fUIInRtStatHide(ADR(tyP0932MagConv3.tyFB.tyBtnRemoteUnclamp.uiMaskRtStat));
		fUIInRtStatHide(ADR(tyP0932MagConv3.tyFB.tyBtnSelClamp.uiMaskRtStat));
		fUIInRtStatHide(ADR(tyP0932MagConv3.tyFB.tyBtnSelUnclamp.uiMaskRtStat));
		fUIInRtStatHide(ADR(tyP0932MagConv3.tyCom.tyBtnSwitch.uiMaskRtStat));

	END_IF
END_IF

	IF p_tyDI.bMagConvCAB717MagSen3 THEN
		fUIInRtStatOff(ADR(tyP0932MagConv3.tyFB.tyBtnSelClamp.uiMaskRtStat));
	END_IF

	IF p_bMagConv2Clp3ClprFixClampCtrl OR p_bMagConv2Clp3ClprRmtClampCtrl THEN
		fUIInRtStatOff(ADR(tyP0932MagConv3.tyFB.tyBtnEnt.uiMaskRtStat));
		fUIInRtStatOff(ADR(tyP0932MagConv3.tyFB.tyBtnExit.uiMaskRtStat));
	END_IF

END_ACTION
```

#### Act_OptP0932MagConv3FBStat.st
```iecst
ACTION Act_OptP0932MagConv3FBStat:

	IF tyP0932MagConv3.tyFB.tyBtnFixedClamp.bValue = TRUE OR tyP0932MagConv3.tyFB.tyBtnRemoteClamp.bValue = TRUE
		OR tyP0932MagConv3.tyFB.tyBtnFixedUnclamp.bValue = TRUE OR tyP0932MagConv3.tyFB.tyBtnRemoteUnclamp.bValue = TRUE
		THEN
		tyP0932MagConv3.tyFB.tyStringStat.sValue	:= p_sMagConv2Clp3StatTxt;
	ELSIF (tyP0932MagConv3.tyFB.tyBtnFixedClamp.bValue = FALSE AND  tyP0932MagConv3.tyFB.tyBtnRemoteClamp.bValue = FALSE
		AND tyP0932MagConv3.tyFB.tyBtnFixedUnclamp.bValue = FALSE AND  tyP0932MagConv3.tyFB.tyBtnRemoteUnclamp.bValue = FALSE
		AND p_eMagConv2Clp3Status <> Busy)
		THEN
		tyP0932MagConv3.tyFB.tyStringStat.sValue	:= p_sMagConv2Clp3StatTxt;

	ELSIF tyP0932MagConv3.tyFB.tyBtnSelUnclamp.bValue = TRUE OR tyP0932MagConv3.tyFB.tyBtnSelClamp.bValue = TRUE
		THEN
		tyP0932MagConv3.tyFB.tyStringStat.sValue	:= p_sSelClamp3StatTxt;
	END_IF
END_ACTION
```

#### Act_OptP0932MagConv3DC.st
```iecst
ACTION Act_OptP0932MagConv3DC:

	//Magazine Conveyor
	IF tyP0932MagConv3.tyDC.tyBtnStop.bRtCompl = TRUE THEN
		eMagConv2Clp3Act	:= MagConv2ClpActStop;

		IF p_eMagConv2Clp3Stat = MagConv2ClpActStop AND p_eMagConv2Clp3Status = Done THEN
			eMagConv2Clp3Act	:= MagConv2ClpActIdle;

			tyP0932MagConv3.tyDC.tyBtnStop.bRtCompl		:= FALSE;
			tyP0932MagConv3.tyDC.tyBtnStop.bValue		:= TRUE;
			tyP0932MagConv3.tyDC.tyBtnStop.bRtLk		:= TRUE;

			tyP0932MagConv3.tyDC.tyBtnMagIn.bRtCompl	:= FALSE;
			tyP0932MagConv3.tyDC.tyBtnMagIn.bValue		:= FALSE;
			tyP0932MagConv3.tyDC.tyBtnMagIn.bRtLk		:= FALSE;

			tyP0932MagConv3.tyDC.tyBtnMagOut.bRtCompl	:= FALSE;
			tyP0932MagConv3.tyDC.tyBtnMagOut.bValue		:= FALSE;
			tyP0932MagConv3.tyDC.tyBtnMagOut.bRtLk		:= FALSE;
		END_IF

	ELSIF tyP0932MagConv3.tyDC.tyBtnMagIn.bRtCompl = TRUE THEN
		tyP0932MagConv3.tyDC.tyBtnMagIn.bValue	:= TRUE;
		tyP0932MagConv3.tyDC.tyBtnMagIn.bRtLk	:= TRUE;

		tyP0932MagConv3.tyDC.tyBtnStop.bValue	:= FALSE;
		tyP0932MagConv3.tyDC.tyBtnStop.bRtLk	:= FALSE;

		IF p_tyNtParamCurr.eProjMagConvDir = ConvDirLToR OR p_tyNtParamCurr.eProjMagConvDir = ConvDirLToL THEN

			eMagConv2Clp3Act	:= MagConv2ClpActSetMtrSigOnOrLToR;

			IF p_eMagConv2Clp3Stat = MagConv2ClpActSetMtrSigOnOrLToR AND p_eMagConv2Clp3Status = Done THEN
				eMagConv2Clp3Act	:= MagConv2ClpActIdle;

				tyP0932MagConv3.tyDC.tyBtnMagIn.bRtCompl	:= FALSE;
			END_IF

		ELSE

			eMagConv2Clp3Act	:= MagConv2ClpActSetMtrDirOrRToL;

			IF p_eMagConv2Clp3Stat = MagConv2ClpActSetMtrDirOrRToL AND p_eMagConv2Clp3Status = Done THEN
				eMagConv2Clp3Act	:= MagConv2ClpActIdle;

				tyP0932MagConv3.tyDC.tyBtnMagIn.bRtCompl	:= FALSE;
			END_IF

		END_IF

	ELSIF tyP0932MagConv3.tyDC.tyBtnMagOut.bRtCompl = TRUE THEN
		tyP0932MagConv3.tyDC.tyBtnMagOut.bValue	:= TRUE;
		tyP0932MagConv3.tyDC.tyBtnMagOut.bRtLk	:= TRUE;

		tyP0932MagConv3.tyDC.tyBtnStop.bValue	:= FALSE;
		tyP0932MagConv3.tyDC.tyBtnStop.bRtLk	:= FALSE;

		IF p_tyNtParamCurr.eProjMagConvDir = ConvDirLToR OR p_tyNtParamCurr.eProjMagConvDir = ConvDirRToR THEN

			eMagConv2Clp3Act	:= MagConv2ClpActSetMtrSigOnOrLToR;

			IF p_eMagConv2Clp3Stat = MagConv2ClpActSetMtrSigOnOrLToR AND p_eMagConv2Clp3Status = Done THEN
				eMagConv2Clp3Act	:= MagConv2ClpActIdle;

				tyP0932MagConv3.tyDC.tyBtnMagOut.bRtCompl	:= FALSE;
			END_IF

		ELSE

			eMagConv2Clp3Act	:= MagConv2ClpActSetMtrDirOrRToL;

			IF p_eMagConv2Clp3Stat = MagConv2ClpActSetMtrDirOrRToL AND p_eMagConv2Clp3Status = Done THEN
				eMagConv2Clp3Act	:= MagConv2ClpActIdle;

				tyP0932MagConv3.tyDC.tyBtnMagOut.bRtCompl	:= FALSE;
			END_IF

		END_IF

	END_IF

	//Magazine Clamper
	IF tyP0932MagConv3.tyCom.tyBtnSwitch.bValue = TRUE THEN
		IF p_bSelClamp3TwoCtrlOut = FALSE THEN
			IF tyP0932MagConv3.tyDC.tyBtnSelUnclamp.bRtCompl = TRUE THEN
				tyP0932MagConv3.tyDC.tyBtnSelUnclamp.bValue := TRUE;
				tyP0932MagConv3.tyDC.tyBtnSelClamp.bValue := FALSE;

				eMagConvSelClp3Act	:= PneuActSetExt;

				IF p_eSelClamp3Stat = PneuActSetExt AND p_eSelClamp3Status = Done THEN
					eMagConvSelClp3Act	:= PneuActIdle;

					tyP0932MagConv3.tyDC.tyBtnSelUnclamp.bRtCompl	:= FALSE;
				END_IF

			ELSIF tyP0932MagConv3.tyDC.tyBtnSelClamp.bRtCompl = TRUE THEN
				tyP0932MagConv3.tyDC.tyBtnSelClamp.bValue := TRUE;
				tyP0932MagConv3.tyDC.tyBtnSelUnclamp.bValue := FALSE;

				eMagConvSelClp3Act	:= PneuActSetRet;

				IF p_eSelClamp3Stat = PneuActSetRet AND p_eSelClamp3Status = Done THEN
					eMagConvSelClp3Act	:= PneuActIdle;

					tyP0932MagConv3.tyDC.tyBtnSelClamp.bRtCompl	:= FALSE;
				END_IF
			END_IF

		ELSE
			IF (tyP0932MagConv3.tyDC.tyBtnSelUnclamp.bRtCompl = TRUE) OR (tyP0932MagConv3.tyDC.tyBtnSelClamp.bRtCompl = TRUE) THEN
				IF (tyP0932MagConv3.tyDC.tyBtnSelUnclamp.bValue = TRUE) AND (tyP0932MagConv3.tyDC.tyBtnSelClamp.bValue = TRUE) THEN
					eMagConvSelClp3Act	:= PneuActSetAll;

					IF p_eSelClamp3Stat = PneuActSetAll AND p_eSelClamp3Status = Done THEN
						eMagConvSelClp3Act	:= PneuActIdle;

						tyP0932MagConv3.tyDC.tyBtnSelUnclamp.bRtCompl		:= FALSE;
						tyP0932MagConv3.tyDC.tyBtnSelClamp.bRtCompl			:= FALSE;
					END_IF

				ELSIF (tyP0932MagConv3.tyDC.tyBtnSelUnclamp.bValue = TRUE) AND (tyP0932MagConv3.tyDC.tyBtnSelClamp.bValue = FALSE) THEN
					eMagConvSelClp3Act	:= PneuActSetExt;

					IF p_eSelClamp3Stat = PneuActSetExt AND p_eSelClamp3Status = Done THEN
						eMagConvSelClp3Act	:= PneuActIdle;

						tyP0932MagConv3.tyDC.tyBtnSelUnclamp.bRtCompl		:= FALSE;
						tyP0932MagConv3.tyDC.tyBtnSelClamp.bRtCompl			:= FALSE;
					END_IF

				ELSIF (tyP0932MagConv3.tyDC.tyBtnSelUnclamp.bValue = FALSE) AND (tyP0932MagConv3.tyDC.tyBtnSelClamp.bValue = TRUE) THEN
					eMagConvSelClp3Act	:= PneuActSetRet;

					IF p_eSelClamp3Stat = PneuActSetRet AND p_eSelClamp3Status = Done THEN
						eMagConvSelClp3Act	:= PneuActIdle;

						tyP0932MagConv3.tyDC.tyBtnSelUnclamp.bRtCompl		:= FALSE;
						tyP0932MagConv3.tyDC.tyBtnSelClamp.bRtCompl			:= FALSE;
					END_IF

				ELSE
					eMagConvSelClp3Act	:= PneuActRstAll;

					IF p_eSelClamp3Stat = PneuActRstAll AND p_eSelClamp3Status = Done THEN
						eMagConvSelClp3Act	:= PneuActIdle;

						tyP0932MagConv3.tyDC.tyBtnSelUnclamp.bRtCompl		:= FALSE;
						tyP0932MagConv3.tyDC.tyBtnSelClamp.bRtCompl			:= FALSE;
					END_IF

				END_IF
			END_IF
		END_IF

		IF p_bMagConv2Clp1ClprTwoOutputCtrl = FALSE THEN

			//Fixed
			IF tyP0932MagConv3.tyDC.tyBtnFixedClamp.bRtCompl = TRUE THEN
				tyP0932MagConv3.tyDC.tyBtnFixedClamp.bValue		:= TRUE;
				tyP0932MagConv3.tyDC.tyBtnFixedUnclamp.bValue	:= FALSE;

				eMagConv2Clp3Act	:= MagConv2ClpActFixClprSetClamp;

				IF p_eMagConv2Clp3Stat = MagConv2ClpActFixClprSetClamp AND p_eMagConv2Clp3Status = Done THEN
					eMagConv2Clp3Act	:= MagConv2ClpActIdle;

					tyP0932MagConv3.tyDC.tyBtnFixedClamp.bRtCompl	:= FALSE;
				END_IF

			ELSIF tyP0932MagConv3.tyDC.tyBtnFixedUnclamp.bRtCompl = TRUE THEN
				tyP0932MagConv3.tyDC.tyBtnFixedUnclamp.bValue	:= TRUE;
				tyP0932MagConv3.tyDC.tyBtnFixedClamp.bValue		:= FALSE;

				eMagConv2Clp3Act	:= MagConv2ClpActFixClprSetUnclamp;

				IF p_eMagConv2Clp3Stat = MagConv2ClpActFixClprSetUnclamp AND p_eMagConv2Clp3Status = Done THEN
					eMagConv2Clp3Act	:= MagConv2ClpActIdle;

					tyP0932MagConv3.tyDC.tyBtnFixedUnclamp.bRtCompl	:= FALSE;
				END_IF

			END_IF

			//Remote
			IF tyP0932MagConv3.tyDC.tyBtnRemoteClamp.bRtCompl = TRUE THEN
				tyP0932MagConv3.tyDC.tyBtnRemoteClamp.bValue		:= TRUE;
				tyP0932MagConv3.tyDC.tyBtnRemoteUnclamp.bValue		:= FALSE;

				eMagConv2Clp3Act	:= MagConv2ClpActRmtClprSetClamp;

				IF p_eMagConv2Clp3Stat = MagConv2ClpActRmtClprSetClamp AND p_eMagConv2Clp3Status = Done THEN
					eMagConv2Clp3Act	:= MagConv2ClpActIdle;

					tyP0932MagConv3.tyDC.tyBtnRemoteClamp.bRtCompl	:= FALSE;
				END_IF

			ELSIF tyP0932MagConv3.tyDC.tyBtnRemoteUnclamp.bRtCompl = TRUE THEN
				tyP0932MagConv3.tyDC.tyBtnRemoteUnclamp.bValue	:= TRUE;
				tyP0932MagConv3.tyDC.tyBtnRemoteClamp.bValue	:= FALSE;

				eMagConv2Clp3Act	:= MagConv2ClpActRmtClprSetUnclamp;

				IF p_eMagConv2Clp3Stat = MagConv2ClpActRmtClprSetUnclamp AND p_eMagConv2Clp3Status = Done THEN
					eMagConv2Clp3Act	:= MagConv2ClpActIdle;

					tyP0932MagConv3.tyDC.tyBtnRemoteUnclamp.bRtCompl	:= FALSE;
				END_IF

			END_IF

		ELSE

			//Fixed
			IF (tyP0932MagConv3.tyDC.tyBtnFixedClamp.bRtCompl = TRUE) OR (tyP0932MagConv3.tyDC.tyBtnFixedUnclamp.bRtCompl = TRUE) THEN

				IF (tyP0932MagConv3.tyDC.tyBtnFixedClamp.bValue = TRUE) AND (tyP0932MagConv3.tyDC.tyBtnFixedUnclamp.bValue = TRUE) THEN

					eMagConv2Clp3Act	:= MagConv2ClpActFixClprSetAll;

					IF p_eMagConv2Clp3Stat = MagConv2ClpActFixClprSetAll AND p_eMagConv2Clp3Status = Done THEN

						eMagConv2Clp3Act	:= MagConv2ClpActIdle;

						tyP0932MagConv3.tyDC.tyBtnFixedClamp.bRtCompl	:= FALSE;
						tyP0932MagConv3.tyDC.tyBtnFixedUnclamp.bRtCompl	:= FALSE;
					END_IF

				ELSIF (tyP0932MagConv3.tyDC.tyBtnFixedClamp.bValue = TRUE) AND (tyP0932MagConv3.tyDC.tyBtnFixedUnclamp.bValue = FALSE) THEN
					eMagConv2Clp3Act	:= MagConv2ClpActFixClprSetClamp;

					IF p_eMagConv2Clp3Stat = MagConv2ClpActFixClprSetClamp AND p_eMagConv2Clp3Status = Done THEN

						eMagConv2Clp3Act	:= MagConv2ClpActIdle;

						tyP0932MagConv3.tyDC.tyBtnFixedClamp.bRtCompl	:= FALSE;
						tyP0932MagConv3.tyDC.tyBtnFixedUnclamp.bRtCompl	:= FALSE;
					END_IF

				ELSIF (tyP0932MagConv3.tyDC.tyBtnFixedClamp.bValue = FALSE) AND (tyP0932MagConv3.tyDC.tyBtnFixedUnclamp.bValue = TRUE) THEN
					eMagConv2Clp3Act	:= MagConv2ClpActFixClprSetUnclamp;

					IF p_eMagConv2Clp3Stat = MagConv2ClpActFixClprSetUnclamp AND p_eMagConv2Clp3Status = Done THEN

						eMagConv2Clp3Act	:= MagConv2ClpActIdle;

						tyP0932MagConv3.tyDC.tyBtnFixedClamp.bRtCompl	:= FALSE;
						tyP0932MagConv3.tyDC.tyBtnFixedUnclamp.bRtCompl	:= FALSE;
					END_IF

				ELSE
					eMagConv2Clp3Act	:= MagConv2ClpActFixClprRstAll;

					IF p_eMagConv2Clp3Stat = MagConv2ClpActFixClprRstAll AND p_eMagConv2Clp3Status = Done THEN

						eMagConv2Clp3Act	:= MagConv2ClpActIdle;

						tyP0932MagConv3.tyDC.tyBtnFixedClamp.bRtCompl	:= FALSE;
						tyP0932MagConv3.tyDC.tyBtnFixedUnclamp.bRtCompl	:= FALSE;
					END_IF

				END_IF

				//Remote
				IF (tyP0932MagConv3.tyDC.tyBtnRemoteClamp.bRtCompl = TRUE) OR (tyP0932MagConv3.tyDC.tyBtnRemoteUnclamp.bRtCompl = TRUE) THEN

					IF (tyP0932MagConv3.tyDC.tyBtnRemoteClamp.bValue = TRUE) AND (tyP0932MagConv3.tyDC.tyBtnRemoteUnclamp.bValue = TRUE) THEN

						eMagConv2Clp3Act	:= MagConv2ClpActRmtClprSetAll;

						IF p_eMagConv2Clp3Stat = MagConv2ClpActRmtClprSetAll AND p_eMagConv2Clp3Status = Done THEN

							eMagConv2Clp3Act	:= MagConv2ClpActIdle;

							tyP0932MagConv3.tyDC.tyBtnRemoteClamp.bRtCompl		:= FALSE;
							tyP0932MagConv3.tyDC.tyBtnRemoteUnclamp.bRtCompl	:= FALSE;
						END_IF

					ELSIF (tyP0932MagConv3.tyDC.tyBtnRemoteClamp.bValue = TRUE) AND (tyP0932MagConv3.tyDC.tyBtnRemoteUnclamp.bValue = FALSE) THEN
						eMagConv2Clp3Act	:= MagConv2ClpActRmtClprSetClamp;

						IF p_eMagConv2Clp3Stat = MagConv2ClpActRmtClprSetClamp AND p_eMagConv2Clp3Status = Done THEN

							eMagConv2Clp3Act	:= MagConv2ClpActIdle;

							tyP0932MagConv3.tyDC.tyBtnRemoteClamp.bRtCompl	:= FALSE;
							tyP0932MagConv3.tyDC.tyBtnRemoteUnclamp.bRtCompl	:= FALSE;
						END_IF

					ELSIF (tyP0932MagConv3.tyDC.tyBtnRemoteClamp.bValue = FALSE) AND (tyP0932MagConv3.tyDC.tyBtnRemoteUnclamp.bValue = TRUE) THEN
						eMagConv2Clp3Act	:= MagConv2ClpActRmtClprSetUnclamp;

						IF p_eMagConv2Clp3Stat = MagConv2ClpActRmtClprSetUnclamp AND p_eMagConv2Clp3Status = Done THEN

							eMagConv2Clp3Act	:= MagConv2ClpActIdle;

							tyP0932MagConv3.tyDC.tyBtnRemoteClamp.bRtCompl	:= FALSE;
							tyP0932MagConv3.tyDC.tyBtnRemoteUnclamp.bRtCompl	:= FALSE;
						END_IF

					ELSE
						eMagConv2Clp3Act	:= MagConv2ClpActRmtClprRstAll;

						IF p_eMagConv2Clp3Stat = MagConv2ClpActRmtClprRstAll AND p_eMagConv2Clp3Status = Done THEN

							eMagConv2Clp3Act	:= MagConv2ClpActIdle;

							tyP0932MagConv3.tyDC.tyBtnRemoteClamp.bRtCompl	:= FALSE;
							tyP0932MagConv3.tyDC.tyBtnRemoteUnclamp.bRtCompl	:= FALSE;
						END_IF

					END_IF
				END_IF

			END_IF

		END_IF

		//Fixed
		tyP0932MagConv3.tyFB.tyBtnFixedClamp.bRtCompl		:= FALSE;
		tyP0932MagConv3.tyFB.tyBtnFixedClamp.bValue			:= FALSE;
		tyP0932MagConv3.tyFB.tyBtnFixedUnclamp.bRtCompl		:= FALSE;
		tyP0932MagConv3.tyFB.tyBtnFixedUnclamp.bValue		:= FALSE;

		//Remote
		tyP0932MagConv3.tyFB.tyBtnRemoteClamp.bRtCompl		:= FALSE;
		tyP0932MagConv3.tyFB.tyBtnRemoteClamp.bValue		:= FALSE;
		tyP0932MagConv3.tyFB.tyBtnRemoteUnclamp.bRtCompl	:= FALSE;
		tyP0932MagConv3.tyFB.tyBtnRemoteUnclamp.bValue		:= FALSE;

	END_IF

	//Mask
	IF p_eMagConv2Clp3Status = Error THEN

		fUIInRtStatOff(ADR(tyP0932MagConv3.tyDC.tyBtnMagIn.uiMaskRtStat));
		fUIInRtStatOff(ADR(tyP0932MagConv3.tyDC.tyBtnMagOut.uiMaskRtStat));
		fUIInRtStatOff(ADR(tyP0932MagConv3.tyDC.tyBtnFixedClamp.uiMaskRtStat));
		fUIInRtStatOff(ADR(tyP0932MagConv3.tyDC.tyBtnFixedUnclamp.uiMaskRtStat));
		fUIInRtStatOff(ADR(tyP0932MagConv3.tyDC.tyBtnRemoteClamp.uiMaskRtStat));
		fUIInRtStatOff(ADR(tyP0932MagConv3.tyDC.tyBtnRemoteUnclamp.uiMaskRtStat));

	ELSIF tyP0932MagConv3.tyDC.tyBtnMagIn.bValue = TRUE THEN

		fUIInRtStatHide(ADR(tyP0932MagConv3.tyDC.tyBtnMagIn.uiMaskRtStat));
		fUIInRtStatOff(ADR(tyP0932MagConv3.tyDC.tyBtnMagOut.uiMaskRtStat));
		fUIInRtStatOff(ADR(tyP0932MagConv3.tyDC.tyBtnFixedClamp.uiMaskRtStat));
		fUIInRtStatOff(ADR(tyP0932MagConv3.tyDC.tyBtnFixedUnclamp.uiMaskRtStat));
		fUIInRtStatOff(ADR(tyP0932MagConv3.tyDC.tyBtnRemoteClamp.uiMaskRtStat));
		fUIInRtStatOff(ADR(tyP0932MagConv3.tyDC.tyBtnRemoteUnclamp.uiMaskRtStat));

	ELSIF tyP0932MagConv3.tyDC.tyBtnMagOut.bValue = TRUE THEN

		fUIInRtStatOff(ADR(tyP0932MagConv3.tyDC.tyBtnMagIn.uiMaskRtStat));
		fUIInRtStatHide(ADR(tyP0932MagConv3.tyDC.tyBtnMagOut.uiMaskRtStat));
		fUIInRtStatOff(ADR(tyP0932MagConv3.tyDC.tyBtnFixedClamp.uiMaskRtStat));
		fUIInRtStatOff(ADR(tyP0932MagConv3.tyDC.tyBtnFixedUnclamp.uiMaskRtStat));
		fUIInRtStatOff(ADR(tyP0932MagConv3.tyDC.tyBtnRemoteClamp.uiMaskRtStat));
		fUIInRtStatOff(ADR(tyP0932MagConv3.tyDC.tyBtnRemoteUnclamp.uiMaskRtStat));

	ELSE

		fUIInRtStatHide(ADR(tyP0932MagConv3.tyDC.tyBtnMagIn.uiMaskRtStat));
		fUIInRtStatHide(ADR(tyP0932MagConv3.tyDC.tyBtnMagOut.uiMaskRtStat));
		fUIInRtStatHide(ADR(tyP0932MagConv3.tyDC.tyBtnFixedClamp.uiMaskRtStat));
		fUIInRtStatHide(ADR(tyP0932MagConv3.tyDC.tyBtnFixedUnclamp.uiMaskRtStat));
		fUIInRtStatHide(ADR(tyP0932MagConv3.tyDC.tyBtnRemoteClamp.uiMaskRtStat));
		fUIInRtStatHide(ADR(tyP0932MagConv3.tyDC.tyBtnRemoteUnclamp.uiMaskRtStat));

	END_IF

END_ACTION
```

#### Act_OptP0932RstMnl.st
```iecst
ACTION Act_OptP0932RstMnl:

	IF EDGEPOS((bManualMod = FALSE) OR (p_eMagConv2Clp3Status = Error)) THEN

		eMagConv2Clp3Act	:= MagConv2ClpActIdle;
		eMagConvSelClp3Act	:= PneuActIdle;
		//Magazine Conveyor
		//FB
		tyP0932MagConv3.tyFB.tyBtnEnt.bRtCompl				:= FALSE;
		tyP0932MagConv3.tyFB.tyBtnExit.bRtCompl				:= FALSE;
		tyP0932MagConv3.tyFB.tyBtnStop.bRtCompl				:= FALSE;

		tyP0932MagConv3.tyFB.tyBtnEnt.bValue				:= FALSE;
		tyP0932MagConv3.tyFB.tyBtnExit.bValue				:= FALSE;
		tyP0932MagConv3.tyFB.tyBtnStop.bValue				:= TRUE;

		tyP0932MagConv3.tyFB.tyBtnEnt.bRtLk					:= FALSE;
		tyP0932MagConv3.tyFB.tyBtnExit.bRtLk				:= FALSE;
		tyP0932MagConv3.tyFB.tyBtnStop.bRtLk				:= TRUE;

		tyP0932MagConv3.tyFB.tyBtnEnt.uiMaskRtStat.0		:= TRUE;
		tyP0932MagConv3.tyFB.tyBtnExit.uiMaskRtStat.0		:= TRUE;
		tyP0932MagConv3.tyCom.tyBtnSwitch.uiMaskRtStat.0	:= TRUE;

		//Direct
		tyP0932MagConv3.tyDC.tyBtnMagIn.bRtCompl			:= FALSE;
		tyP0932MagConv3.tyDC.tyBtnMagOut.bRtCompl			:= FALSE;
		tyP0932MagConv3.tyDC.tyBtnStop.bRtCompl				:= FALSE;

		tyP0932MagConv3.tyDC.tyBtnMagIn.bValue				:= FALSE;
		tyP0932MagConv3.tyDC.tyBtnMagOut.bValue				:= FALSE;
		tyP0932MagConv3.tyDC.tyBtnStop.bValue				:= TRUE;

		tyP0932MagConv3.tyDC.tyBtnMagIn.bRtLk				:= FALSE;
		tyP0932MagConv3.tyDC.tyBtnMagOut.bRtLk				:= FALSE;
		tyP0932MagConv3.tyDC.tyBtnStop.bRtLk				:= TRUE;

		tyP0932MagConv3.tyDC.tyBtnMagIn.uiMaskRtStat.0		:= TRUE;
		tyP0932MagConv3.tyDC.tyBtnMagOut.uiMaskRtStat.0		:= TRUE;
		tyP0932MagConv3.tyCom.tyBtnSwitch.uiMaskRtStat.0	:= TRUE;

		//Magazine Clamper
		//FB
		//Fixed
		tyP0932MagConv3.tyFB.tyBtnFixedClamp.bRtCompl			:= FALSE;
		tyP0932MagConv3.tyFB.tyBtnFixedUnclamp.bRtCompl			:= FALSE;

		tyP0932MagConv3.tyFB.tyBtnFixedClamp.bValue				:= FALSE;
		tyP0932MagConv3.tyFB.tyBtnFixedUnclamp.bValue			:= FALSE;

		//Remote
		tyP0932MagConv3.tyFB.tyBtnRemoteClamp.bRtCompl			:= FALSE;
		tyP0932MagConv3.tyFB.tyBtnRemoteUnclamp.bRtCompl		:= FALSE;

		tyP0932MagConv3.tyFB.tyBtnRemoteClamp.bValue			:= FALSE;
		tyP0932MagConv3.tyFB.tyBtnRemoteUnclamp.bValue			:= FALSE;

		//Selection
		tyP0932MagConv3.tyFB.tyBtnSelClamp.bRtCompl			:= FALSE;
		tyP0932MagConv3.tyFB.tyBtnSelUnclamp.bRtCompl		:= FALSE;

		tyP0932MagConv3.tyFB.tyBtnSelClamp.bValue			:= FALSE;
		tyP0932MagConv3.tyFB.tyBtnSelUnclamp.bValue			:= FALSE;

		tyP0932MagConv3.tyFB.tyBtnFixedClamp.uiMaskRtStat.0		:= TRUE;
		tyP0932MagConv3.tyFB.tyBtnFixedUnclamp.uiMaskRtStat.0	:= TRUE;
		tyP0932MagConv3.tyFB.tyBtnRemoteClamp.uiMaskRtStat.0	:= TRUE;
		tyP0932MagConv3.tyFB.tyBtnRemoteUnclamp.uiMaskRtStat.0	:= TRUE;
		tyP0932MagConv3.tyFB.tyBtnSelClamp.uiMaskRtStat.0		:= TRUE;
		tyP0932MagConv3.tyFB.tyBtnSelUnclamp.uiMaskRtStat.0		:= TRUE;

		tyP0932MagConv3.tyCom.tyBtnSwitch.uiMaskRtStat.0		:= TRUE;

		//Direct
		//Fixed
		tyP0932MagConv3.tyDC.tyBtnFixedClamp.bRtCompl			:= FALSE;
		tyP0932MagConv3.tyDC.tyBtnFixedUnclamp.bRtCompl			:= FALSE;

		tyP0932MagConv3.tyDC.tyBtnFixedClamp.bValue				:= FALSE;
		tyP0932MagConv3.tyDC.tyBtnFixedUnclamp.bValue			:= FALSE;

		//Remote
		tyP0932MagConv3.tyDC.tyBtnRemoteClamp.bRtCompl			:= FALSE;
		tyP0932MagConv3.tyDC.tyBtnRemoteUnclamp.bRtCompl		:= FALSE;

		tyP0932MagConv3.tyDC.tyBtnRemoteClamp.bValue			:= FALSE;
		tyP0932MagConv3.tyDC.tyBtnRemoteUnclamp.bValue			:= FALSE;

		//Selection
		tyP0932MagConv3.tyDC.tyBtnSelClamp.bRtCompl				:= FALSE;
		tyP0932MagConv3.tyDC.tyBtnSelUnclamp.bRtCompl			:= FALSE;

		tyP0932MagConv3.tyDC.tyBtnSelClamp.bValue				:= FALSE;
		tyP0932MagConv3.tyDC.tyBtnSelUnclamp.bValue				:= FALSE;

		tyP0932MagConv3.tyDC.tyBtnFixedClamp.uiMaskRtStat.0		:= TRUE;
		tyP0932MagConv3.tyDC.tyBtnFixedUnclamp.uiMaskRtStat.0	:= TRUE;
		tyP0932MagConv3.tyDC.tyBtnRemoteClamp.uiMaskRtStat.0	:= TRUE;
		tyP0932MagConv3.tyDC.tyBtnRemoteUnclamp.uiMaskRtStat.0	:= TRUE;
		tyP0932MagConv3.tyDC.tyBtnSelClamp.uiMaskRtStat.0		:= TRUE;
		tyP0932MagConv3.tyDC.tyBtnSelUnclamp.uiMaskRtStat.0		:= TRUE;

		tyP0932MagConv3.tyCom.tyBtnSwitch.uiMaskRtStat.0		:= TRUE;

	END_IF

	IF EDGEPOS(bManualMod = FALSE) THEN
		tyP0932MagConv3.tyCom.tyBtnSwitch.bValue := FALSE;

		IF p_tyNtParamCurr.bMagAutoVerifyPrep = FALSE THEN
			fUIInRtStatHide(ADR(tyP0932MagConv3.tyDC.tyLyrWithoutSelClamp.uiRtStat));
			fUIInRtStatOff(ADR(tyP0932MagConv3.tyFB.tyLyrWithoutSelClamp.uiRtStat));
		ELSE

			fUIInRtStatHide(ADR(tyP0932MagConv3.tyDC.tyLyr.uiRtStat));
			fUIInRtStatOff(ADR(tyP0932MagConv3.tyFB.tyLyr.uiRtStat));
		END_IF
	END_IF

END_ACTION
```

#### Act_EntP0933Disp.st
```iecst
ACTION Act_EntP0933Disp:

	//Access Address
	p_tyC0002FullMask ACCESS ADR(tyP0933PushConv.tyFullMaskHide);

	p_tyC0004Navi ACCESS ADR(tyP0933PushConv.tyNaviBack);

	p_tyC0005Main ACCESS ADR(tyCommon.tyMain);

	p_tyC0007Notif ACCESS ADR(tyCommon.tyNotif);

	p_tyC0008MsgBox ACCESS ADR(tyP0933PushConv.tyMsgBoxHide);

	p_tyC0009Info ACCESS ADR(tyCommon.tyInfo);

	p_tyP0933PushConvCom ACCESS ADR(tyP0933PushConv.tyCom);
	p_tyP0933PushConvDC ACCESS ADR(tyP0933PushConv.tyDC);
	p_tyP0933PushlConvFB ACCESS ADR(tyP0933PushConv.tyFB);

	//Display
	tyP0933PushConv.tyFB.tyNumExtSpd.diValue			:= p_tyProdRcpCurrRcp0.diMtrPshrExtSpd;
	tyP0933PushConv.tyFB.tyNumExtTorqPercent.diValue	:= p_tyProdRcpCurrRcp0.diMtrPshrExtTorq;

END_ACTION
```

#### Act_OptP0933Navi.st
```iecst
ACTION Act_OptP0933Navi:

	IF tyP0933PushConv.tyNaviBack.tyBtnBack.bRtCompl = TRUE THEN
		eChgPage		:= UIP0920MtrNPneuCtrl;

		tyP0933PushConv.tyNaviBack.tyBtnBack.bRtCompl		:= FALSE;
		tyP0933PushConv.tyNaviBack.tyBtnBack.bValue			:= FALSE;
	END_IF

END_ACTION
```

#### Act_OptP0933FullMask.st
```iecst
ACTION Act_OptP0933FullMask:

	IF eCurrPage = UIP0933PusherConv THEN

		IF p_tyDI.bEStopSig = FALSE THEN
			p_tyC0002FullMask ACCESS ADR(tyP0933PushConv.tyFullMaskEStop);

		ELSIF p_tyDI.bCoverSWSig = FALSE THEN
			p_tyC0002FullMask ACCESS ADR(tyP0933PushConv.tyFullMaskCWSig);

		ELSIF p_tyDI.bSafetyRlySig = FALSE THEN
			p_tyC0002FullMask ACCESS ADR(tyP0933PushConv.tyFullMaskSafetyRly);

		ELSIF p_tyNtParamCurr.bProjOutletShutPrep AND
			(p_tyDI.bOutShutterOpenRS = FALSE AND ((ABS(p_diTravActualPos - p_tyMagRcpCurrRcp.diMag1TravPosInUM) < 500) OR p_bTravIsHomed = FALSE))
			OR (p_tyDI.bOutShutterOpenRS2 = FALSE AND ((ABS(p_diTravActualPos - p_tyMagRcpCurrRcp.diMag2TravPosInUM) < 500) OR p_bTravIsHomed = FALSE))
			OR (p_tyDI.bOutShutterOpenRS3 = FALSE AND ((ABS(p_diTravActualPos - p_tyMagRcpCurrRcp.diMag3TravPosInUM) < 500) OR p_bTravIsHomed = FALSE)) THEN

			//	p_tyC0002FullMask ACCESS ADR(tyP0933PushConv.tyFullMaskOutShutterInterrupt);
			p_tyC0002FullMask ACCESS ADR(tyP0933PushConv.tyFullMaskHide);
			tyP0933PushConv.tyCom.tyTxtExtWarning.sValue := sPshrExtWarnMsg;
			tyP0933PushConv.tyCom.tyTxtExtWarning.uiRtStat := FALSE;

		ELSIF p_tyNtParamCurr.bAWPrep AND  p_tyNtParamCurr.bAWPusherPrep
			AND p_tyMcParamCurr.bAWDis = FALSE
			AND p_bAWOpenIsHomed = FALSE
			AND (p_diAWPushOrPullerActualPos + p_tyMcParamCurr.diAWPusherAtHmPosInUM )>(p_tyMcParamCurr.diWidthAtHmPosInUM - p_diAWOpenActualPos-15000)
			THEN
			p_tyC0002FullMask ACCESS ADR(tyP0933PushConv.tyFullMaskAWConvInterrupt);

		ELSE
			p_tyC0002FullMask ACCESS ADR(tyP0933PushConv.tyFullMaskHide);
			tyP0933PushConv.tyCom.tyTxtExtWarning.uiRtStat := TRUE;

		END_IF

	END_IF

END_ACTION
```

#### Act_OptP0933Keypad.st
```iecst
ACTION Act_OptP0933Keypad:

	IF fUIOutRtStatTPIsOpen(ADR(tyP0933PullConv.tyFB.tyNumExtSpd.uiRtStat)) = TRUE THEN
		tyProperty.tyKeypad.tyStringTitle.sKeypadTitle	:= tyP0933PushConv.tyFB.tyNumExtSpd.sKeypadTitle;

	ELSIF fUIOutRtStatTPIsOpen(ADR(tyP0933PullConv.tyFB.tyNumExtTorqPercent.uiRtStat)) = TRUE THEN
		tyProperty.tyKeypad.tyStringTitle.sKeypadTitle	:= tyP0933PushConv.tyFB.tyNumExtTorqPercent.sKeypadTitle;

	END_IF

END_ACTION
```

#### Act_OptP0933PusherConvChgLyr.st
```iecst
ACTION Act_OptP0933PusherConvChgLyr:

	IF tyP0933PushConv.tyCom.tyBtnSwitch.bRtCompl THEN
		tyP0933PushConv.tyCom.tyBtnSwitch.bRtCompl := FALSE;
		IF tyP0933PushConv.tyCom.tyBtnSwitch.bValue = TRUE THEN
			fUIInRtStatOff(ADR(tyP0933PushConv.tyDC.tyLyr.uiRtStat));
			fUIInRtStatHide(ADR(tyP0933PushConv.tyFB.tyLyr.uiRtStat));
		ELSE
			fUIInRtStatHide(ADR(tyP0933PushConv.tyDC.tyLyr.uiRtStat));
			fUIInRtStatOff(ADR(tyP0933PushConv.tyFB.tyLyr.uiRtStat));
		END_IF

	END_IF

	//Mask
	IF tyP0933PushConv.tyFB.tyBtnExt.bRtCompl OR tyP0933PushConv.tyFB.tyBtnRet.bRtCompl OR tyP0933PushConv.tyFB.tyBtnStop.bRtCompl
		OR tyP0933PushConv.tyDC.tyBtnAlarmRst.bValue OR tyP0933PushConv.tyDC.tyBtnBrake.bValue OR tyP0933PushConv.tyDC.tyBtnExt.bValue OR tyP0933PushConv.tyDC.tyBtnRet.bValue OR tyP0933PushConv.tyDC.tyBtnSigOn.bValue OR tyP0933PushConv.tyDC.tyBtnSpdBinBit0.bValue OR tyP0933PushConv.tyDC.tyBtnSpdBinBit1.bValue OR tyP0933PushConv.tyDC.tyBtnSpdBinBit2.bValue THEN

		fUIInRtStatOff(ADR(tyP0933PushConv.tyCom.tyBtnSwitch.uiMaskRtStat));
	ELSE
		fUIInRtStatHide(ADR(tyP0933PushConv.tyCom.tyBtnSwitch.uiMaskRtStat));
	END_IF

END_ACTION
```

#### Act_OptP0933PusherConvSen.st
```iecst
ACTION Act_OptP0933PusherConvSen:

	tyP0933PushConv.tyCom.tyBtnLftSen.bValue	:= p_tyDI.bConvLftSen;
	tyP0933PushConv.tyCom.tyBtnMidSen.bValue	:= p_tyDI.bConvMidSen;
	tyP0933PushConv.tyCom.tyBtnRgtSen.bValue	:= p_tyDI.bConvRgtSen;
	tyP0933PushConv.tyCom.tyBtnClrSen.bValue	:= p_tyDI.bConvClrSen;
	tyP0933PushConv.tyCom.tyBtnExtRS.bValue		:= p_tyDI.bPusherExtRS;
	tyP0933PushConv.tyCom.tyBtnRetRS.bValue		:= p_tyDI.bPusherRetRS;

	tyP0933PushConv.tyCom.tyBtnExtSlwSen.bValue	:= p_tyDI.bPusherExtSlwSen;
	tyP0933PushConv.tyCom.tyBtnRetSlwSen.bValue	:= p_tyDI.bPusherRetSlwSen;

	tyP0933PushConv.tyCom.tyBtnAlarmSig.bValue	:= p_tyDI.bMtrPshrAlmSig;
	tyP0933PushConv.tyCom.tyBtnTorqueSig.bValue	:= p_tyDI.bMtrPshrTorqueSig;

	tyP0933PushConv.tyCom.tyBtnAntiJamSen.bValue := p_tyDI.bPshrAntiJam;

	//Machine Bitmap
	IF tyP0933PushConv.tyFB.tyBtnExt.bRtCompl OR tyP0933PushConv.tyDC.tyBtnExt.bRtCompl THEN

		tyP0933PushConv.tyCom.tyBitmapMc.uiValueIdx	:= 2;

	ELSIF tyP0933PushConv.tyFB.tyBtnRet.bRtCompl OR tyP0933PushConv.tyDC.tyBtnRet.bRtCompl THEN

		tyP0933PushConv.tyCom.tyBitmapMc.uiValueIdx	:= 1;

	ELSIF tyP0933PushConv.tyFB.tyBtnCylExit.bRtCompl OR tyP0933PushConv.tyFB.tyBtnEnt.bRtCompl OR tyP0933PushConv.tyFB.tyBtnExit.bRtCompl OR tyP0933PushConv.tyFB.tyBtnStop.bRtCompl
		OR tyP0933PushConv.tyDC.tyBtnStart.bRtCompl OR tyP0933PushConv.tyDC.tyBtnStop.bRtCompl THEN

		tyP0933PushConv.tyCom.tyBitmapMc.uiValueIdx	:= 0;

	END_IF

	IF p_tyNtParamCurr.eProjMag = ULMagTriple AND p_tyNtParamCurr.bMagAutoVerifyPrep = TRUE AND p_tyNtParamCurr.bProjMotorizedPusherPrep = FALSE THEN
		IF 	tyP0933PushConv.tyCom.tyBitmapMc.uiValueIdx < 100 THEN
			tyP0933PushConv.tyCom.tyBitmapMc.uiValueIdx	:= tyP0933PushConv.tyCom.tyBitmapMc.uiValueIdx + 100;
		END_IF
	ELSIF p_tyNtParamCurr.eProjMag = ULMagTriple AND p_tyNtParamCurr.bMagAutoVerifyPrep = FALSE AND p_tyNtParamCurr.bProjMotorizedPusherPrep = TRUE THEN
			IF 	tyP0933PushConv.tyCom.tyBitmapMc.uiValueIdx < 400 THEN
				tyP0933PushConv.tyCom.tyBitmapMc.uiValueIdx	:= tyP0933PushConv.tyCom.tyBitmapMc.uiValueIdx + 400;
		END_IF
	END_IF

END_ACTION
```
